(* CoDeSys 2.3.9.25 project: 1.pro *)
(* Libraries: ifm_CR0200\ifm_CR0200_DUMMY_V060002.lib 18.5.06 14:18:58, D:\program files\ifm electronic\CoDeSys V2.3\Targets\ifm\Library\ifm_hydraulic_16bitOS04_V010001.lib 23.10.09 15:40:02, ifm_CR0200\ifm_CR0200_V060003.lib 5.11.09 16:13:42, standard.lib 4.10.05 11:14:46, SysLibCallback.lib 5.6.03 00:36:48, 3S_CANopenManagerOptTableEx.lib 16.7.10 11:11:06, 3S_CanDrvOptTableEx.lib 16.7.10 11:11:16, 3S_CANopenNetVarOptTableEx.lib 16.7.10 11:11:26, Util.lib 6.11.07 14:39:24, ifm_CR0200\ifm_CR0200_CANopenMaster_V040003.lib 7.2.07 16:08:18, 3S_CANopenMasterOptTableEx.lib 16.7.10 11:11:12 *)

(* PLC configuration (modules and I/O channels)
Inputs/Outputs [CR0200] node 0, in %IB0 out %QB0
  Inputs Port0 [Eingangsport0] node 0, in %IB0 out %QB0
    I00 AT %IX0.0 [BoolChannelIn] Connector 1, Pin 08, (see Configuration Byte I00_MODE)
    I01 AT %IX0.1 [BoolChannelIn] Connector 1, Pin 27, (see Configuration Byte I01_MODE)
    I02 AT %IX0.2 [BoolChannelIn] Connector 1, Pin 09, (see Configuration Byte I02_MODE)
    I03 AT %IX0.3 [BoolChannelIn] Connector 1, Pin 28, (see Configuration Byte I03_MODE)
    I04 AT %IX0.4 [BoolChannelIn] Connector 1, Pin 10, (see Configuration Byte I04_MODE)
    I05 AT %IX0.5 [BoolChannelIn] Connector 1, Pin 29, (see Configuration Byte I05_MODE)
    I06 AT %IX0.6 [BoolChannelIn] Connector 1, Pin 11, (see Configuration Byte I06_MODE)
    I07 AT %IX0.7 [BoolChannelIn] Connector 1, Pin 30, (see Configuration Byte I07_MODE)
  Inputs Port1 [Eingangsport1] node 0, in %IB1 out %QB0
    I10 AT %IX0.8 [BoolChannelIn] Connector 1, Pin 44, (see Configuration Byte I10_MODE)
    I11 AT %IX0.9 [BoolChannelIn] Connector 1, Pin 45, (see Configuration Byte I11_MODE)
    I12 AT %IX0.10 [BoolChannelIn] Connector 1, Pin 46, (see Configuration Byte I12_MODE)
    I13 AT %IX0.11 [BoolChannelIn] Connector 1, Pin 47, (see Configuration Byte I13_MODE)
    I14 AT %IX0.12 [BoolChannelIn] Connector 1, Pin 20, (see Configuration Byte I14_MODE)
    I15 AT %IX0.13 [BoolChannelIn] Connector 1, Pin 02, (see Configuration Byte I15_MODE)
    I16 AT %IX0.14 [BoolChannelIn] Connector 1, Pin 21, (see Configuration Byte I16_MODE)
    I17 AT %IX0.15 [BoolChannelIn] Connector 1, Pin 38, (see Configuration Byte I17_MODE)
  Inputs Port2 [Eingangsport2] node 0, in %IB2 out %QB0
    I20 AT %IX1.0 [BoolChannelIn] Connector 1, Pin 36, (see Configuration Byte I20_MODE)
    I21 AT %IX1.1 [BoolChannelIn] Connector 1, Pin 54, (see Configuration Byte I21_MODE)
    I22 AT %IX1.2 [BoolChannelIn] Connector 1, Pin 17, (see Configuration Byte I22_MODE)
    I23 AT %IX1.3 [BoolChannelIn] Connector 1, Pin 53, (see Configuration Byte I23_MODE)
    I24 AT %IX1.4 [BoolChannelIn] Connector 1, Pin 19, (see Configuration Byte I24_MODE)
    I25 AT %IX1.5 [BoolChannelIn] Connector 1, Pin 55, (see Configuration Byte I25_MODE)
    I26 AT %IX1.6 [BoolChannelIn] Connector 1, Pin 18, (see Configuration Byte I26_MODE)
    I27 AT %IX1.7 [BoolChannelIn] Connector 1, Pin 37, (see Configuration Byte I27_MODE)
  Inputs Port3 [Eingangsport3] node 0, in %IB3 out %QB0
    I30 AT %IX1.8 [BoolChannelIn] Connector 1, Pin 39, (see Configuration Byte I30_MODE)
    I31 AT %IX1.9 [BoolChannelIn] Connector 1, Pin 03, (see Configuration Byte I31_MODE)
    I32 AT %IX1.10 [BoolChannelIn] Connector 1, Pin 40, (see Configuration Byte I32_MODE)
    I33 AT %IX1.11 [BoolChannelIn] Connector 1, Pin 22, (see Configuration Byte I33_MODE)
    I34 AT %IX1.12 [BoolChannelIn] Connector 1, Pin 41, (see Configuration Byte I34_MODE)
    I35 AT %IX1.13 [BoolChannelIn] Connector 1, Pin 42, (see Configuration Byte I35_MODE)
    I36 AT %IX1.14 [BoolChannelIn] Connector 1, Pin 43, (see Configuration Byte I36_MODE)
    I37 AT %IX1.15 [BoolChannelIn] Connector 1, Pin 04, (see Configuration Byte I37_MODE)
  Inputs Port4 [Eingangsport4] node 0, in %IB4 out %QB0
    I40 AT %IX2.0 [BoolChannelIn] Connector 1, Pin 48, (see Configuration Byte I40_MODE)
    I41 AT %IX2.1 [BoolChannelIn] Connector 1, Pin 49, (see Configuration Byte I41_MODE)
    I42 AT %IX2.2 [BoolChannelIn] Connector 1, Pin 31, (see Configuration Byte I42_MODE)
    I43 AT %IX2.3 [BoolChannelIn] Connector 1, Pin 50, (see Configuration Byte I43_MODE)
    I44 AT %IX2.4 [BoolChannelIn] Connector 1, Pin 51, (see Configuration Byte I44_MODE)
    I45 AT %IX2.5 [BoolChannelIn] Connector 1, Pin 52, (see Configuration Byte I45_MODE)
    I46 AT %IX2.6 [BoolChannelIn] Connector 1, Pin 16, (see Configuration Byte I46_MODE)
    I47 AT %IX2.7 [BoolChannelIn] Connector 1, Pin 35, (see Configuration Byte I47_MODE)
  Inputs Analog [Analogport] node 0, in %IB6 out %QB0
    ANALOG0 AT %IW3 [WordChannelIn] Connector 1, Pin 08, ANALOG CHANNEL 0
    ANALOG1 AT %IW4 [WordChannelIn] Connector 1, Pin 27, ANALOG CHANNEL 1
    ANALOG2 AT %IW5 [WordChannelIn] Connector 1, Pin 09, ANALOG CHANNEL 2
    ANALOG3 AT %IW6 [WordChannelIn] Connector 1, Pin 28, ANALOG CHANNEL 3
    ANALOG4 AT %IW7 [WordChannelIn] Connector 1, Pin 10, ANALOG CHANNEL 4
    ANALOG5 AT %IW8 [WordChannelIn] Connector 1, Pin 29, ANALOG CHANNEL 5
    ANALOG6 AT %IW9 [WordChannelIn] Connector 1, Pin 11, ANALOG CHANNEL 6
    ANALOG7 AT %IW10 [WordChannelIn] Connector 1, Pin 30, ANALOG CHANNEL 7
  Inputs Miscellaneous [Eingaenge] node 0, in %IB22 out %QB0
    SUPPLY_VOLTAGE AT %IW11 [WordChannelIn] SUPPLY VOLTAGE
    CLAMP_15 AT %IX12.0 [WordChannelIn] CLAMP 15
  Outputs Port1 [Ausgangsport1] node 0, in %IB64 out %QB0
    Q10 AT %QX0.0 [BoolChannelOut] Connector 1, Pin 44, (see Configuration Byte Q10_MODE)
    Q11 AT %QX0.1 [BoolChannelOut] Connector 1, Pin 45, (see Configuration Byte Q11_MODE)
    Q12 AT %QX0.2 [BoolChannelOut] Connector 1, Pin 46, (see Configuration Byte Q12_MODE)
    Q13 AT %QX0.3 [BoolChannelOut] Connector 1, Pin 47, (see Configuration Byte Q13_MODE)
  Outputs Port2 [Ausgangsport2] node 0, in %IB64 out %QB0
    Q20 AT %QX0.4 [BoolChannelOut] Connector 1, Pin 36, (see Configuration Byte Q20_MODE)
    Q21 AT %QX0.5 [BoolChannelOut] Connector 1, Pin 54, (see Configuration Byte Q21_MODE)
    Q22 AT %QX0.6 [BoolChannelOut] Connector 1, Pin 17, (see Configuration Byte Q22_MODE)
    Q23 AT %QX0.7 [BoolChannelOut] Connector 1, Pin 53, (see Configuration Byte Q23_MODE)
  Outputs Port3 [Ausgangsport3] node 0, in %IB64 out %QB1
    Q30 AT %QX0.8 [BoolChannelOut] Connector 1, Pin 39, (see Configuration Byte Q30_MODE)
    Q31 AT %QX0.9 [BoolChannelOut] Connector 1, Pin 03, (see Configuration Byte Q31_MODE)
    Q32 AT %QX0.10 [BoolChannelOut] Connector 1, Pin 40, (see Configuration Byte Q32_MODE)
    Q33 AT %QX0.11 [BoolChannelOut] Connector 1, Pin 22, (see Configuration Byte Q33_MODE)
    Q34 AT %QX0.12 [BoolChannelOut] Connector 1, Pin 41, (see Configuration Byte Q34_MODE)
    Q35 AT %QX0.13 [BoolChannelOut] Connector 1, Pin 42, (see Configuration Byte Q35_MODE)
    Q36 AT %QX0.14 [BoolChannelOut] Connector 1, Pin 43, (see Configuration Byte Q36_MODE)
    Q37 AT %QX0.15 [BoolChannelOut] Connector 1, Pin 04, (see Configuration Byte Q37_MODE)
  Outputs Port4 [Ausgangsport4] node 0, in %IB64 out %QB2
    Q40 AT %QX1.0 [BoolChannelOut] Connector 1, Pin 48, (see Configuration Byte Q40_MODE)
    Q41 AT %QX1.1 [BoolChannelOut] Connector 1, Pin 49, (see Configuration Byte Q41_MODE)
    Q42 AT %QX1.2 [BoolChannelOut] Connector 1, Pin 31, (see Configuration Byte Q42_MODE)
    Q43 AT %QX1.3 [BoolChannelOut] Connector 1, Pin 50, (see Configuration Byte Q43_MODE)
    Q44 AT %QX1.4 [BoolChannelOut] Connector 1, Pin 51, (see Configuration Byte Q44_MODE)
    Q45 AT %QX1.5 [BoolChannelOut] Connector 1, Pin 52, (see Configuration Byte Q45_MODE)
    Q46 AT %QX1.6 [BoolChannelOut] Connector 1, Pin 16, (see Configuration Byte Q46_MODE)
    Q47 AT %QX1.7 [BoolChannelOut] Connector 1, Pin 35, (see Configuration Byte Q47_MODE)
  Input Modes Port0 [EingangsModi0] node 0, in %IB64 out %QB8
    I00_MODE AT %QB8 [ByteChannelOut] Configuration Byte for Input Pin 08, Connector 1
    I01_MODE AT %QB9 [ByteChannelOut] Configuration Byte for Input Pin 27, Connector 1
    I02_MODE AT %QB10 [ByteChannelOut] Configuration Byte for Input Pin 09, Connector 1
    I03_MODE AT %QB11 [ByteChannelOut] Configuration Byte for Input Pin 28, Connector 1
    I04_MODE AT %QB12 [ByteChannelOut] Configuration Byte for Input Pin 10, Connector 1
    I05_MODE AT %QB13 [ByteChannelOut] Configuration Byte for Input Pin 29, Connector 1
    I06_MODE AT %QB14 [ByteChannelOut] Configuration Byte for Input Pin 11, Connector 1
    I07_MODE AT %QB15 [ByteChannelOut] Configuration Byte for Input Pin 30, Connector 1
  Input Modes Port1 [EingangsModi1] node 0, in %IB64 out %QB16
    I14_MODE AT %QB16 [ByteChannelOut] Configuration Byte for Input Pin 20, Connector 1
    I15_MODE AT %QB17 [ByteChannelOut] Configuration Byte for Input Pin 02, Connector 1
    I16_MODE AT %QB18 [ByteChannelOut] Configuration Byte for Input Pin 21, Connector 1
    I17_MODE AT %QB19 [ByteChannelOut] Configuration Byte for Input Pin 38, Connector 1
  Input Modes Port2 [EingangsModi2] node 0, in %IB64 out %QB20
    I24_MODE AT %QB20 [ByteChannelOut] Configuration Byte for Input Pin 19, Connector 1
    I25_MODE AT %QB21 [ByteChannelOut] Configuration Byte for Input Pin 55, Connector 1
    I26_MODE AT %QB22 [ByteChannelOut] Configuration Byte for Input Pin 18, Connector 1
    I27_MODE AT %QB23 [ByteChannelOut] Configuration Byte for Input Pin 37, Connector 1
  Input Modes Port3 [EingangsModi3] node 0, in %IB64 out %QB24
    I30_MODE AT %QB24 [ByteChannelOut] Configuration Byte for Input Pin 39, Connector 1
    I31_MODE AT %QB25 [ByteChannelOut] Configuration Byte for Input Pin 03, Connector 1
    I32_MODE AT %QB26 [ByteChannelOut] Configuration Byte for Input Pin 40, Connector 1
    I33_MODE AT %QB27 [ByteChannelOut] Configuration Byte for Input Pin 22, Connector 1
    I34_MODE AT %QB28 [ByteChannelOut] Configuration Byte for Input Pin 41, Connector 1
    I35_MODE AT %QB29 [ByteChannelOut] Configuration Byte for Input Pin 42, Connector 1
    I36_MODE AT %QB30 [ByteChannelOut] Configuration Byte for Input Pin 43, Connector 1
    I37_MODE AT %QB31 [ByteChannelOut] Configuration Byte for Input Pin 04, Connector 1
  Input Modes Port4 [EingangsModi4] node 0, in %IB64 out %QB32
    I40_MODE AT %QB32 [ByteChannelOut] Configuration Byte for Input Pin 48, Connector 1
    I41_MODE AT %QB33 [ByteChannelOut] Configuration Byte for Input Pin 49, Connector 1
    I42_MODE AT %QB34 [ByteChannelOut] Configuration Byte for Input Pin 31, Connector 1
    I43_MODE AT %QB35 [ByteChannelOut] Configuration Byte for Input Pin 50, Connector 1
    I44_MODE AT %QB36 [ByteChannelOut] Configuration Byte for Input Pin 51, Connector 1
    I45_MODE AT %QB37 [ByteChannelOut] Configuration Byte for Input Pin 52, Connector 1
    I46_MODE AT %QB38 [ByteChannelOut] Configuration Byte for Input Pin 16, Connector 1
    I47_MODE AT %QB39 [ByteChannelOut] Configuration Byte for Input Pin 35, Connector 1
  Output Modes Port1 [AusgangsModi1] node 0, in %IB64 out %QB40
    Q10_MODE AT %QB40 [ByteChannelOut] Configuration Byte for Output Pin 44, Connector 1
    Q11_MODE AT %QB41 [ByteChannelOut] Configuration Byte for Output Pin 45, Connector 1
    Q12_MODE AT %QB42 [ByteChannelOut] Configuration Byte for Output Pin 46, Connector 1
    Q13_MODE AT %QB43 [ByteChannelOut] Configuration Byte for Output Pin 47, Connector 1
  Output Modes Port2 [AusgangsModi2] node 0, in %IB64 out %QB44
    Q20_MODE AT %QB44 [ByteChannelOut] Configuration Byte for Output Pin 36, Connector 1
    Q21_MODE AT %QB45 [ByteChannelOut] Configuration Byte for Output Pin 54, Connector 1
    Q22_MODE AT %QB46 [ByteChannelOut] Configuration Byte for Output Pin 17, Connector 1
    Q23_MODE AT %QB47 [ByteChannelOut] Configuration Byte for Output Pin 53, Connector 1
  Output Modes Port3 [AusgangsModi3] node 0, in %IB64 out %QB48
    Q30_MODE AT %QB48 [ByteChannelOut] Configuration Byte for Output Pin 39, Connector 1
    Q31_MODE AT %QB49 [ByteChannelOut] Configuration Byte for Output Pin 03, Connector 1
    Q32_MODE AT %QB50 [ByteChannelOut] Configuration Byte for Output Pin 40, Connector 1
    Q33_MODE AT %QB51 [ByteChannelOut] Configuration Byte for Output Pin 22, Connector 1
    Q34_MODE AT %QB52 [ByteChannelOut] Configuration Byte for Output Pin 41, Connector 1
    Q35_MODE AT %QB53 [ByteChannelOut] Configuration Byte for Output Pin 42, Connector 1
    Q36_MODE AT %QB54 [ByteChannelOut] Configuration Byte for Output Pin 43, Connector 1
    Q37_MODE AT %QB55 [ByteChannelOut] Configuration Byte for Output Pin 04, Connector 1
  Output Modes Port4 [AusgangsModi4] node 0, in %IB64 out %QB56
    Q40_MODE AT %QB56 [ByteChannelOut] Configuration Byte for Output Pin 48, Connector 1
    Q41_MODE AT %QB57 [ByteChannelOut] Configuration Byte for Output Pin 49, Connector 1
    Q42_MODE AT %QB58 [ByteChannelOut] Configuration Byte for Output Pin 31, Connector 1
    Q43_MODE AT %QB59 [ByteChannelOut] Configuration Byte for Output Pin 50, Connector 1
    Q44_MODE AT %QB60 [ByteChannelOut] Configuration Byte for Output Pin 51, Connector 1
    Q45_MODE AT %QB61 [ByteChannelOut] Configuration Byte for Output Pin 52, Connector 1
    Q46_MODE AT %QB62 [ByteChannelOut] Configuration Byte for Output Pin 16, Connector 1
    Q47_MODE AT %QB63 [ByteChannelOut] Configuration Byte for Output Pin 35, Connector 1
Extended Inputs Port0 [Eingangsport0E] node 0, in %IB64 out %QB64
  I00_E AT %IX32.0 [BoolChannelIn] Connector 2, Pin 08, (see Configuration Byte I00_MODE_E)
  I01_E AT %IX32.1 [BoolChannelIn] Connector 2, Pin 27, (see Configuration Byte I01_MODE_E)
  I02_E AT %IX32.2 [BoolChannelIn] Connector 2, Pin 09, (see Configuration Byte I02_MODE_E)
  I03_E AT %IX32.3 [BoolChannelIn] Connector 2, Pin 28, (see Configuration Byte I03_MODE_E)
  I04_E AT %IX32.4 [BoolChannelIn] Connector 2, Pin 10, (see Configuration Byte I04_MODE_E)
  I05_E AT %IX32.5 [BoolChannelIn] Connector 2, Pin 29, (see Configuration Byte I05_MODE_E)
  I06_E AT %IX32.6 [BoolChannelIn] Connector 2, Pin 11, (see Configuration Byte I06_MODE_E)
  I07_E AT %IX32.7 [BoolChannelIn] Connector 2, Pin 30, (see Configuration Byte I07_MODE_E)
Extended Inputs Port1 [Eingangsport1E] node 0, in %IB65 out %QB64
  I10_E AT %IX32.8 [BoolChannelIn] Connector 2, Pin 44, (see Configuration Byte I10_MODE_E)
  I11_E AT %IX32.9 [BoolChannelIn] Connector 2, Pin 45, (see Configuration Byte I11_MODE_E)
  I12_E AT %IX32.10 [BoolChannelIn] Connector 2, Pin 46, (see Configuration Byte I12_MODE_E)
  I13_E AT %IX32.11 [BoolChannelIn] Connector 2, Pin 47, (see Configuration Byte I13_MODE_E)
  I14_E AT %IX32.12 [BoolChannelIn] Connector 2, Pin 20, (see Configuration Byte I14_MODE_E)
  I15_E AT %IX32.13 [BoolChannelIn] Connector 2, Pin 02, (see Configuration Byte I15_MODE_E)
  I16_E AT %IX32.14 [BoolChannelIn] Connector 2, Pin 21, (see Configuration Byte I16_MODE_E)
  I17_E AT %IX32.15 [BoolChannelIn] Connector 2, Pin 38, (see Configuration Byte I17_MODE_E)
I20_E AT %IX33.0 [BoolChannelIn] Connector 2, Pin 36, (see Configuration Byte I20_MODE_E)
I21_E AT %IX33.1 [BoolChannelIn] Connector 2, Pin 54, (see Configuration Byte I21_MODE_E)
I22_E AT %IX33.2 [BoolChannelIn] Connector 2, Pin 17, (see Configuration Byte I22_MODE_E)
I23_E AT %IX33.3 [BoolChannelIn] Connector 2, Pin 53, (see Configuration Byte I23_MODE_E)
I24_E AT %IX33.4 [BoolChannelIn] Connector 2, Pin 19, (see Configuration Byte I24_MODE_E)
I25_E AT %IX33.5 [BoolChannelIn] Connector 2, Pin 55, (see Configuration Byte I25_MODE_E)
I26_E AT %IX33.6 [BoolChannelIn] Connector 2, Pin 18, (see Configuration Byte I26_MODE_E)
I27_E AT %IX33.7 [BoolChannelIn] Connector 2, Pin 37, (see Configuration Byte I27_MODE_E)
I30_E AT %IX33.8 [BoolChannelIn] Connector 2, Pin 39, (see Configuration Byte I30_MODE_E)
I31_E AT %IX33.9 [BoolChannelIn] Connector 2, Pin 03, (see Configuration Byte I31_MODE_E)
I32_E AT %IX33.10 [BoolChannelIn] Connector 2, Pin 40, (see Configuration Byte I32_MODE_E)
I33_E AT %IX33.11 [BoolChannelIn] Connector 2, Pin 22, (see Configuration Byte I33_MODE_E)
I34_E AT %IX33.12 [BoolChannelIn] Connector 2, Pin 41, (see Configuration Byte I34_MODE_E)
I35_E AT %IX33.13 [BoolChannelIn] Connector 2, Pin 42, (see Configuration Byte I35_MODE_E)
I36_E AT %IX33.14 [BoolChannelIn] Connector 2, Pin 43, (see Configuration Byte I36_MODE_E)
I37_E AT %IX33.15 [BoolChannelIn] Connector 2, Pin 04, (see Configuration Byte I37_MODE_E)
Extended Inputs Port4 [Eingangsport4E] node 0, in %IB68 out %QB64
  I40_E AT %IX34.0 [BoolChannelIn] Connector 2, Pin 48, (see Configuration Byte I40_MODE_E)
  I41_E AT %IX34.1 [BoolChannelIn] Connector 2, Pin 49, (see Configuration Byte I41_MODE_E)
  I42_E AT %IX34.2 [BoolChannelIn] Connector 2, Pin 31, (see Configuration Byte I42_MODE_E)
  I43_E AT %IX34.3 [BoolChannelIn] Connector 2, Pin 50, (see Configuration Byte I43_MODE_E)
  I44_E AT %IX34.4 [BoolChannelIn] Connector 2, Pin 51, (see Configuration Byte I44_MODE_E)
  I45_E AT %IX34.5 [BoolChannelIn] Connector 2, Pin 52, (see Configuration Byte I45_MODE_E)
  I46_E AT %IX34.6 [BoolChannelIn] Connector 2, Pin 16, (see Configuration Byte I46_MODE_E)
  I47_E AT %IX34.7 [BoolChannelIn] Connector 2, Pin 35, (see Configuration Byte I47_MODE_E)
Extended Inputs Analog [AnalogportE] node 0, in %IB70 out %QB64
  ANALOG0_E AT %IW35 [WordChannelIn] Connector 2, Pin 08, ANALOG CHANNEL 0
  ANALOG1_E AT %IW36 [WordChannelIn] Connector 2, Pin 27, ANALOG CHANNEL 1
  ANALOG2_E AT %IW37 [WordChannelIn] Connector 2, Pin 09, ANALOG CHANNEL 2
  ANALOG3_E AT %IW38 [WordChannelIn] Connector 2, Pin 28, ANALOG CHANNEL 3
  ANALOG4_E AT %IW39 [WordChannelIn] Connector 2, Pin 10, ANALOG CHANNEL 4
  ANALOG5_E AT %IW40 [WordChannelIn] Connector 2, Pin 29, ANALOG CHANNEL 5
  ANALOG6_E AT %IW41 [WordChannelIn] Connector 2, Pin 11, ANALOG CHANNEL 6
  ANALOG7_E AT %IW42 [WordChannelIn] Connector 2, Pin 30, ANALOG CHANNEL 7
Extended Inputs Miscellaneous [EingaengeE] node 0, in %IB86 out %QB64
  SUPPLY_VOLTAGE_E AT %IW43 [WordChannelIn] SUPPLY VOLTAGE
  CLAMP_15_E AT %IX44.0 [WordChannelIn] CLAMP 15
Extended Outputs Port1 [Ausgangsport1E] node 0, in %IB128 out %QB64
  Q10_E AT %QX32.0 [BoolChannelOut] Connector 2, Pin 44, (see Configuration Byte Q10_MODE_E)
  Q11_E AT %QX32.1 [BoolChannelOut] Connector 2, Pin 45, (see Configuration Byte Q11_MODE_E)
  Q12_E AT %QX32.2 [BoolChannelOut] Connector 2, Pin 46, (see Configuration Byte Q11_MODE_E)
  Q13_E AT %QX32.3 [BoolChannelOut] Connector 2, Pin 47, (see Configuration Byte Q11_MODE_E)
Extended Outputs Port2 [Ausgangsport2E] node 0, in %IB128 out %QB64
  Q20_E AT %QX32.4 [BoolChannelOut] Connector 2, Pin 36, (see Configuration Byte Q20_MODE_E)
  Q21_E AT %QX32.5 [BoolChannelOut] Connector 2, Pin 54, (see Configuration Byte Q21_MODE_E)
  Q22_E AT %QX32.6 [BoolChannelOut] Connector 2, Pin 17, (see Configuration Byte Q22_MODE_E)
  Q23_E AT %QX32.7 [BoolChannelOut] Connector 2, Pin 53, (see Configuration Byte Q23_MODE_E)
Q30_E AT %QX32.8 [BoolChannelOut] Connector 2, Pin 39, (see Configuration Byte Q30_MODE_E)
Q31_E AT %QX32.9 [BoolChannelOut] Connector 2, Pin 03, (see Configuration Byte Q31_MODE_E)
Q32_E AT %QX32.10 [BoolChannelOut] Connector 2, Pin 40, (see Configuration Byte Q32_MODE_E)
Q33_E AT %QX32.11 [BoolChannelOut] Connector 2, Pin 22, (see Configuration Byte Q33_MODE_E)
Q34_E AT %QX32.12 [BoolChannelOut] Connector 2, Pin 41, (see Configuration Byte Q34_MODE_E)
Q35_E AT %QX32.13 [BoolChannelOut] Connector 2, Pin 42, (see Configuration Byte Q35_MODE_E)
Q36_E AT %QX32.14 [BoolChannelOut] Connector 2, Pin 43, (see Configuration Byte Q36_MODE_E)
Q37_E AT %QX32.15 [BoolChannelOut] Connector 2, Pin 04, (see Configuration Byte Q37_MODE_E)
Extended Outputs Port4 [Ausgangsport4E] node 0, in %IB128 out %QB66
  Q40_E AT %QX33.0 [BoolChannelOut] Connector 2, Pin 48, (see Configuration Byte Q40_MODE_E)
  Q41_E AT %QX33.1 [BoolChannelOut] Connector 2, Pin 49, (see Configuration Byte Q41_MODE_E)
  Q42_E AT %QX33.2 [BoolChannelOut] Connector 2, Pin 31, (see Configuration Byte Q42_MODE_E)
  Q43_E AT %QX33.3 [BoolChannelOut] Connector 2, Pin 50, (see Configuration Byte Q43_MODE_E)
  Q44_E AT %QX33.4 [BoolChannelOut] Connector 2, Pin 51, (see Configuration Byte Q44_MODE_E)
  Q45_E AT %QX33.5 [BoolChannelOut] Connector 2, Pin 52, (see Configuration Byte Q45_MODE_E)
  Q46_E AT %QX33.6 [BoolChannelOut] Connector 2, Pin 16, (see Configuration Byte Q46_MODE_E)
  Q47_E AT %QX33.7 [BoolChannelOut] Connector 2, Pin 35, (see Configuration Byte Q47_MODE_E)
Extended Input Modes Port0 [EingangsModi0E] node 0, in %IB128 out %QB72
  I00Mode_E AT %QB72 [ByteChannelOut] Configuration Byte for Input Pin 08, Connector 2
  I01Mode_E AT %QB73 [ByteChannelOut] Configuration Byte for Input Pin 27, Connector 2
  I02Mode_E AT %QB74 [ByteChannelOut] Configuration Byte for Input Pin 09, Connector 2
  I03Mode_E AT %QB75 [ByteChannelOut] Configuration Byte for Input Pin 28, Connector 2
  I04Mode_E AT %QB76 [ByteChannelOut] Configuration Byte for Input Pin 10, Connector 2
  I05Mode_E AT %QB77 [ByteChannelOut] Configuration Byte for Input Pin 29, Connector 2
  I06Mode_E AT %QB78 [ByteChannelOut] Configuration Byte for Input Pin 11, Connector 2
  I07Mode_E AT %QB79 [ByteChannelOut] Configuration Byte for Input Pin 30, Connector 2
Extended Input Modes Port1 [EingangsModi1E] node 0, in %IB128 out %QB80
  I14Mode_E AT %QB80 [ByteChannelOut] Configuration Byte for Input Pin 20, Connector 2
  I15Mode_E AT %QB81 [ByteChannelOut] Configuration Byte for Input Pin 02, Connector 2
  I16Mode_E AT %QB82 [ByteChannelOut] Configuration Byte for Input Pin 21, Connector 2
  I17Mode_E AT %QB83 [ByteChannelOut] Configuration Byte for Input Pin 38, Connector 2
Extended Input Modes Port2 [EingangsModi2E] node 0, in %IB128 out %QB84
  I24Mode_E AT %QB84 [ByteChannelOut] Configuration Byte for Input Pin 19, Connector 2
  I25Mode_E AT %QB85 [ByteChannelOut] Configuration Byte for Input Pin 55, Connector 2
  I26Mode_E AT %QB86 [ByteChannelOut] Configuration Byte for Input Pin 18, Connector 2
  I27Mode_E AT %QB87 [ByteChannelOut] Configuration Byte for Input Pin 37, Connector 2
Extended Input Modes Port3 [EingangsModi3E] node 0, in %IB128 out %QB88
  I30Mode_E AT %QB88 [ByteChannelOut] Configuration Byte for Input Pin 39, Connector 2
  I31Mode_E AT %QB89 [ByteChannelOut] Configuration Byte for Input Pin 03, Connector 2
  I32Mode_E AT %QB90 [ByteChannelOut] Configuration Byte for Input Pin 40, Connector 2
  I33Mode_E AT %QB91 [ByteChannelOut] Configuration Byte for Input Pin 22, Connector 2
  I34Mode_E AT %QB92 [ByteChannelOut] Configuration Byte for Input Pin 41, Connector 2
  I35Mode_E AT %QB93 [ByteChannelOut] Configuration Byte for Input Pin 42, Connector 2
  I36Mode_E AT %QB94 [ByteChannelOut] Configuration Byte for Input Pin 43, Connector 2
  I37Mode_E AT %QB95 [ByteChannelOut] Configuration Byte for Input Pin 04, Connector 2
Extended Input Modes Port4 [EingangsModi4E] node 0, in %IB128 out %QB96
  I40Mode_E AT %QB96 [ByteChannelOut] Configuration Byte for Input Pin 48, Connector 2
  I41Mode_E AT %QB97 [ByteChannelOut] Configuration Byte for Input Pin 49, Connector 2
  I42Mode_E AT %QB98 [ByteChannelOut] Configuration Byte for Input Pin 31, Connector 2
  I43Mode_E AT %QB99 [ByteChannelOut] Configuration Byte for Input Pin 50, Connector 2
  I44Mode_E AT %QB100 [ByteChannelOut] Configuration Byte for Input Pin 51, Connector 2
  I45Mode_E AT %QB101 [ByteChannelOut] Configuration Byte for Input Pin 52, Connector 2
  I46Mode_E AT %QB102 [ByteChannelOut] Configuration Byte for Input Pin 16, Connector 2
  I47Mode_E AT %QB103 [ByteChannelOut] Configuration Byte for Input Pin 35, Connector 2
Extended Output Modes Port1 [AusgangsModi1E] node 0, in %IB128 out %QB104
  Q10Mode_E AT %QB104 [ByteChannelOut] Configuration Byte for Output Pin 44, Connector 2
  Q11Mode_E AT %QB105 [ByteChannelOut] Configuration Byte for Output Pin 45, Connector 2
  Q12Mode_E AT %QB106 [ByteChannelOut] Configuration Byte for Output Pin 46, Connector 2
  Q13Mode_E AT %QB107 [ByteChannelOut] Configuration Byte for Output Pin 47, Connector 2
Extended Output Modes Port2 [AusgangsModi2E] node 0, in %IB128 out %QB108
  Q20Mode_E AT %QB108 [ByteChannelOut] Configuration Byte for Output Pin 36, Connector 2
  Q21Mode_E AT %QB109 [ByteChannelOut] Configuration Byte for Output Pin 54, Connector 2
  Q22Mode_E AT %QB110 [ByteChannelOut] Configuration Byte for Output Pin 17, Connector 2
  Q23Mode_E AT %QB111 [ByteChannelOut] Configuration Byte for Output Pin 53, Connector 2
Extended Output Modes Port3 [AusgangsModi3E] node 0, in %IB128 out %QB112
  Q30Mode_E AT %QB112 [ByteChannelOut] Configuration Byte for Output Pin 39, Connector 2
  Q31Mode_E AT %QB113 [ByteChannelOut] Configuration Byte for Output Pin 03, Connector 2
  Q32Mode_E AT %QB114 [ByteChannelOut] Configuration Byte for Output Pin 40, Connector 2
  Q33Mode_E AT %QB115 [ByteChannelOut] Configuration Byte for Output Pin 22, Connector 2
  Q34Mode_E AT %QB116 [ByteChannelOut] Configuration Byte for Output Pin 41, Connector 2
  Q35Mode_E AT %QB117 [ByteChannelOut] Configuration Byte for Output Pin 42, Connector 2
  Q36Mode_E AT %QB118 [ByteChannelOut] Configuration Byte for Output Pin 43, Connector 2
  Q37Mode_E AT %QB119 [ByteChannelOut] Configuration Byte for Output Pin 04, Connector 2
Extended Output Modes Port4 [AusgangsModi4E] node 0, in %IB128 out %QB120
  Q40Mode_E AT %QB120 [ByteChannelOut] Configuration Byte for Output Pin 48, Connector 2
  Q41Mode_E AT %QB121 [ByteChannelOut] Configuration Byte for Output Pin 49, Connector 2
  Q42Mode_E AT %QB122 [ByteChannelOut] Configuration Byte for Output Pin 31, Connector 2
  Q43Mode_E AT %QB123 [ByteChannelOut] Configuration Byte for Output Pin 50, Connector 2
  Q44Mode_E AT %QB124 [ByteChannelOut] Configuration Byte for Output Pin 51, Connector 2
  Q45Mode_E AT %QB125 [ByteChannelOut] Configuration Byte for Output Pin 52, Connector 2
  Q46Mode_E AT %QB126 [ByteChannelOut] Configuration Byte for Output Pin 16, Connector 2
  Q47Mode_E AT %QB127 [ByteChannelOut] Configuration Byte for Output Pin 35, Connector 2
CR0200, CANopen Master [CanMaster] node 2, in %IB192 out %QB192
*)

(* Global variable list: alarm/alarm_text *)
VAR_GLOBAL

	mv_alarm10001:			BOOL;
	mv_alarm10002:			BOOL;
	mv_alarm10003:			BOOL;
	mv_alarm10004:			BOOL;
	mv_alarm10005: 			BOOL;
	mv_alarm10006: 			BOOL;
	mv_alarm10007: 			BOOL;
	mv_alarm10008:			BOOL;

	mv_alarm10009:			BOOL;
	mv_alarm10010:			BOOL;
	mv_alarm10011:			BOOL;
	mv_alarm10012:			BOOL;
	mv_alarm10013:			BOOL;
	mv_alarm10014: 			BOOL;
	mv_alarm10015: 			BOOL;
	mv_alarm10016: 			BOOL;

	mv_alarm10017:			BOOL;
	mv_alarm10018:			BOOL;
	mv_alarm10019:			BOOL;
	mv_alarm10020:			BOOL;
	mv_alarm10021:			BOOL;
	mv_alarm10022: 			BOOL;
	mv_alarm10023: 			BOOL;
	mv_alarm10024: 			BOOL;

	mv_alarm10025:			BOOL;
	mv_alarm10026:			BOOL;
	mv_alarm10027:			BOOL;
	mv_alarm10028:			BOOL;
	mv_alarm10029:			BOOL;
	mv_alarm10030: 			BOOL;
	mv_alarm10031: 			BOOL;
	mv_alarm10032: 			BOOL;
END_VAR

(* Global variable list: CanOpen implicit Variables *)
VAR_GLOBAL CONSTANT
	MAX_CTRLINDEX : INT := 0;
END_VAR
VAR_GLOBAL CONSTANT
	USE_CANOPEN_NODES : BOOL := FALSE;
	MAX_MASTERINDEX : INT := 0;
	MAX_NODEINDEX : INT := 0;
	MAX_SDOINDEX : INT := 0;
	MAX_PDOINDEX_RX : INT := 0;
	MAX_PDOINDEX_TX : INT := 0;
	MAX_MASTER_ODENTRY_IDX : INT := 0;
END_VAR
VAR_GLOBAL
	pCANopenMaster : ARRAY[0..MAX_MASTERINDEX] OF CanOpenMaster;
	pCanOpenNode : ARRAY[0..MAX_NODEINDEX] OF CanOpenNode;
	pCanOpenSDO : ARRAY[0..MAX_SDOINDEX] OF CanOpenSDO;
	pCanOpenPDO_Rx : ARRAY[0..MAX_PDOINDEX_RX] OF CanOpenPDO_Rx;
	pCanOpenPDO_Tx : ARRAY[0..MAX_PDOINDEX_TX] OF CanOpenPDO_Tx;
	 ODMEntries: ARRAY[0..MAX_MASTER_ODENTRY_IDX] OF CanOpenODEntry;
END_VAR

(* Global variable list: Globale_Variablen *)
VAR_GLOBAL RETAIN
	leveled							:BOOL:=0;
(***通用版程序选择***)
(*
	YT32		10000
	YT32A		10001
	YT32B		10002
	YT32C		10003
	YT32D		10004
	YT32E		10005
	YT32F		10006
	YT32G		10007
	YT32H		10008
	YT32I		10009
	YT32J		10010
	YT32K		10011
	YT32L		10012
	YT32M		10013
	YT32N		10014
	YT32O		10015
	YT32P		10016
	YT32Q		10017
	YT32R		10018
	YT32S		10019
	YT32T		10020
*)
	vehicle_styel					: INT:=10012;
END_VAR

VAR_GLOBAL
	Code_1key					:BOOL;
	Speed_value					:BYTE;
	speed_l						:BOOL;
	encod_sign					: BYTE;
	encod_udint					: UDINT;
	turn_desk_angle				: INT;
(***全局变量***)
	boot_set						: BOOL;
	frequ_set						:BOOL:=1;
	valve_act						: BOOL;

	head_f							:BOOL;
	head_b						:BOOL;
	head_f2						:BOOL;
	head_b2						:BOOL;
	head_f3						:BOOL;
	head_b3						:BOOL;

	auto_extend_triger				: BOOL;
	auto_drawback_triger				: BOOL;

	work_speed_l					:INT;
	work_speed_h				:INT;
	low_speed_l					:INT;
	low_speed_h					:INT;
	high_speed_l					:INT;
	high_speed_h				:INT;

	cruise_sign_set				:BOOL;

	angle_danger01				: INT :=500;
	angle_danger02				: INT := 1500;

	init_1							: BOOL:=TRUE;
	extend_step					:INT;
	withdraw_step				: INT;

	angle_x_offset 				AT%MW0		:INT:=952;
	angle_y_offset 				AT%MW2		:INT:=1039;
	water_height_sign_L 			AT%MW4		: INT:=480;
	water_height_sign_H 		AT%MW6		: INT:=1557;
	oil_pressure_0				AT%MW8		: INT:=4000;
	oil_pressure_22				AT%MW10		: INT:=13931;
	foam_height_sign_L			AT%MW12		: INT:=480;
	foam_height_sign_H			AT%MW14		: INT:=1557;
	water_pressure_0			AT%MW16		: INT:=4000;
	water_pressure_6			AT%MW18		: INT:=6300;

	extend_do						:BOOL;
	withdraw_do					:BOOL;
	high_speed_set				:BOOL;
	high_speed_set1				:BOOL;


 	 extend_left_lv_triger_act		:BOOL;
	extend_right_lv_triger_act	:BOOL;

	rl_ys							:INT:=8;

	triger_left_ground_for			:INT;

	angle_x_m					: WORD;(*倾角X轴实测*)
	angle_y_m					: WORD;(*倾角Y轴实测*)
	oil_pressure_m				: WORD;(*油压实测*)

(***支腿遥控器变量***)
	remote_manual_alarm				:BOOL;
	remote_not_arm_to_station_alarm	:BOOL;

(***网络变量***)
	speed_m						:REAL;
	down_com_sign				:BOOL;
	beep_signal					:BOOL;

	stage_extend_do				:BOOL;
	stage_draw_do				:BOOL;
(***转台变量***)
	tt_turn_com					:BOOL;
	tt_emergency_pump			:BOOL;

	up_down_switch				:BOOL;
	tt_foot_switch					:BOOL;
	tt_engine_startup				:BOOL;
	tt_engine_stop				:BOOL;
	tt_water_pump_open		 	:BOOL;

	tt_engine_acc					:BOOL;(*发动机加速*)
	tt_engine_dec					:BOOL;(*发动机减速*)

	tt_water_canon_open	 		:BOOL;
	tt_water_canon_close	 	:BOOL;

(***工作斗变量***)
	sudden_pump_button		:BOOL;
	stage_extend_over			:BOOL;
	stage_draw_over				:BOOL;

	stage_foot_switch			:BOOL;
	stage_engine_startup		:BOOL;
	stage_engine_stop			:BOOL;
	stage_water_pump_open	:BOOL;
	stage_com					:BOOL;
	stage_engine_acc			:BOOL;(*发动机加速*)
	stage_engine_dec			:BOOL;(*发动机减速*)
	error1							:BOOL;
	error2							:BOOL;

(***屏幕变量***)

	foam_low_sign_set			:BOOL;
	foam_high_sign_set			:BOOL;
	down_zero_set				:BOOL;
	water_low_sign_set			:BOOL;
	water_high_sign_set			:BOOL;
	oil_low_sign_set				:BOOL;
	oil_high_sign_set				:BOOL;
	water_alarm_c				:BOOL;

END_VAR

(* Global variable list: VEHICLE TYPE/io_Variables *)
VAR_GLOBAL
(*************************************A_INPUT*******************************************)
	angle_x												: INT;		(*倾角X轴*)
	angle_y												: INT;		(*倾角Y轴*)
	angle_x_1												: INT;
	angle_y_1												: INT;
	oil_pressure											: WORD;	(*油压*)
	water_pressure										: WORD;	(*系统水压*)
	water_height_sign									: WORD;	(*水位信号*)
	foam_height_sign									: WORD;	(*泡沫液位信号*)
	water_flux												: WORD;	(*水流量信号*)
	speed_sign											: WORD;	(*速度脉冲*)

(**************************************A_OUTPUT***************************************)
	left_front_desired										: WORD;	(*左前垂直伸*)
	right_front_desired									: WORD;	(*右前垂直伸*)
	left_back_desired										: WORD;	(*左后垂直伸*)
	right_back_desired									: WORD;	(*右后垂直伸*)

	right_front_drawback_desired						: WORD;	(*右前垂直收*)
	left_back_drawback_desired							: WORD;	(*左后垂直收*)
	right_back_drawback_desired						: WORD;	(*右后垂直收*)
	left_front_drawback_desired							: WORD;	(*左前垂直收*)

(*************************************D_INPUT*******************************************)
(***支腿***)
	front_left_Lv_ex_check1		(*AT %IX0.6*)			: BOOL;	(*左前水平伸到位*)
	front_right_Lv_ex_check1		(*AT %IX0.7*)			: BOOL;	(*右前水平伸到位*)
	back_left_Lv_ex_check1		(*AT %IX0.12*)		: BOOL;	(*左后水平伸到位*)
	back_right_Lv_ex_check1	(*AT %IX0.13*)		: BOOL;	(*右后水平伸到位*)
	front_left_urt_ex_check1		(*AT %IX0.14*)		: BOOL;	(*左前垂直伸到位*)
	front_right_urt_ex_check1	(*AT %IX0.15*)		: BOOL;	(*右前垂直伸到位*)
	back_left_urt_ex_check1		(*AT %IX1.4*)			: BOOL;	(*左后垂直伸到位*)
	back_right_urt_ex_check1	(*AT %IX1.5*)			: BOOL;	(*右后垂直伸到位*)

	front_left_Lv_ex_check								: BOOL;	(*左前水平伸到位*)
	front_right_Lv_ex_check								: BOOL;	(*右前水平伸到位*)
	back_left_Lv_ex_check								: BOOL;	(*左后水平伸到位*)
	back_right_Lv_ex_check								: BOOL;	(*右后水平伸到位*)
	front_left_urt_ex_check								: BOOL;	(*左前垂直伸到位*)
	front_right_urt_ex_check								: BOOL;	(*右前垂直伸到位*)
	back_left_urt_ex_check								: BOOL;	(*左后垂直伸到位*)
	back_right_urt_ex_check								: BOOL;	(*右后垂直伸到位*)

	front_left_Lv_drb_check		(*AT %IX32.1*)		: BOOL;	(*左前水平收到位*)
	front_right_Lv_drb_check		(*AT %IX32.2*)		: BOOL;	(*右前水平收到位*)
	back_left_Lv_drb_check		(*AT %IX32.3*)		: BOOL;	(*左后水平收到位*)
	back_right_Lv_drb_check	(*AT %IX32.4*)		: BOOL;	(*右后水平收到位*)
	front_left_urt_drb_check1		(*AT %IX32.5*)		: BOOL;	(*左前垂直收到位*)
	front_right_urt_drb_check1	(*AT %IX32.6*)		: BOOL;	(*右前垂直收到位*)
	back_left_urt_drb_check1	(*AT %IX32.7*)		: BOOL;	(*左后垂直收到位*)
	back_right_urt_drb_check1	(*AT %IX32.12	*)		: BOOL;	(*右后垂直收到位*)

	front_left_urt_drb_check								: BOOL;	(*左前垂直收到位*)
	front_right_urt_drb_check							: BOOL;	(*右前垂直收到位*)
	back_left_urt_drb_check								: BOOL;	(*左后垂直收到位*)
	back_right_urt_drb_check							: BOOL;	(*右后垂直收到位*)

(***底盘***)
	engine_run					(*AT %IX2.2*)			: BOOL;	(*发动机启动*)
	engine_stop					(*AT %IX2.3*)			: BOOL;	(*发动机停止*)
	accelerate_sb					(*AT %IX2.0*)			: BOOL;	(*加速*)
	decelerate_sb					(*AT %IX2.1*)			: BOOL;	(*减速*)

(***操作***)
	tt_forcexx						(*AT %IX34.6*)		: BOOL;	(*转台强制*)
	down_force					(*AT %IX34.7*)		: BOOL;	(*下车强制*)
	auto_manu_choice			(*AT %IX34.1*)		: BOOL;	(*自动/手动*)
	water_pump_run_sb			(*AT %IX1.7*)			: BOOL;	(*消防泵开*)
	standby_pump_check								: BOOL;	(*应急泵*)



	left_side_choice 										: BOOL;	(*左单边*)
	right_side_choice										: BOOL;	(*右单边*)

	level_extend_triger_left								: BOOL;	(*自动伸支腿*)
	level_extend_triger_right								: BOOL;	(*自动伸支腿*)
	auto_extend_triger_left								: BOOL;	(*自动伸支腿*)
	auto_extend_triger_right								: BOOL;	(*自动伸支腿*)
	auto_drawback_triger_left							: BOOL;	(*自动收支腿*)
	auto_drawback_triger_right							: BOOL;	(*自动收支腿*)

	level_extend_triger_left1		(*AT %IX34.2*)		: BOOL;	(*自动伸支腿*)
	level_extend_triger_right1	(*AT %IX34.3*)		: BOOL;	(*自动伸支腿*)
	auto_extend_triger_left1		(*AT %IX33.5*)		: BOOL;	(*自动伸支腿*)
	auto_extend_triger_right1	(*AT %IX33.6*)		: BOOL;	(*自动伸支腿*)
	auto_drawback_triger_left1	(*AT %IX33.7*)		: BOOL;	(*自动收支腿*)
	auto_drawback_triger_right1	(*AT %IX34.0*)		: BOOL;	(*自动收支腿*)


(***检测***)
	arm_to_station				(*AT %IX2.4*)			: BOOL;	(*臂架到位检测*)
	water_pump_check			(*AT %IX33.4*)		: BOOL;	(*水泵取力*)
	left_groud_check1			(*AT %IX34.4*)		: BOOL;	(*车胎离地1*)
	left_groud_check2			(*AT %IX34.5*)		: BOOL;	(*车胎离地2*)
	oil_pump_check										: BOOL;	(*油泵检测*)

(***支腿遥控盒***)
	remote_switch_leg									: BOOL;	(*支腿选择*)
	remote_control_left									: BOOL;	(*支腿左*)
	remote_control_right									: BOOL;	(*支腿右*)
	remote_control_up									: BOOL;	(*支腿上*)
	remote_control_down								: BOOL;	(*支腿下*)
	remote_out_front_left									: BOOL;	(*指示灯左前*)
	remote_out_front_back								: BOOL;	(*指示灯左后*)
	remote_out_right_left									: BOOL;	(*指示灯右前*)
	remote_out_right_back								: BOOL;	(*指示灯右后*)

(*************************************D_OUTPUT*****************************************)
(***支腿***)
	left_front_lv_ex_valve			(*AT %QX32.2*)	 	:  BOOL;	(*左前水平伸*)
	left_back_lv_ex_valve			(*AT %QX32.0*) 		:  BOOL;	(*左后水平伸*)
	right_front_lv_ex_valve		(*AT %QX32.6*)		:  BOOL;	(*右前水平伸*)
	right_back_lv_ex_valve		(*AT %QX32.4*)		:  BOOL;	(*右后水平伸*)
	left_front_lv_drb_valve		(*AT %QX32.3*)	 	:  BOOL;	(*左前水平收*)
	left_back_lv_drb_valve		(*AT %QX32.1*) 		:  BOOL;	(*左后水平收*)
	right_front_lv_drb_valve		(*AT %QX32.7*)		:  BOOL;	(*右前水平收*)
	right_back_lv_drb_valve		(*AT %QX32.5*)		:  BOOL;	(*右后水平收*)

(***底盘***)
	enginer_run_ctl				(*AT %QX0.8*)	 		:  BOOL;	(*启动控制*)
	enginer_stop_ctl				(*AT %QX0.9*)	 		:  BOOL;	(*熄火控制*)
	enginer_acc_ctl				(*AT %QX32.9*)	 	:  BOOL;	(*加速控制*)
	enginer_dec_ctl				(*AT %QX32.10*)	 	:  BOOL;	(*减速控制*)

(***操作***)
	water_pump_ctl				(*AT %QX0.10*)	 	:  BOOL;	(*水泵控制*)
	standby_oil_pump							 		:  BOOL;	(*应急泵*)
	up_valve_ctl					(*AT %QX32.14*)	 	:  BOOL;	(*上车阀*)
	down_valve_ctl				(*AT %QX32.15*) 		:  BOOL;	(*下车阀*)

(***指示***)
	over_level_sign				(*AT %QX0.11*)	 	:  BOOL;	(*坡度超限*)
	triger_left_grd_sign			(*AT %QX0.12*)	 	:  BOOL;	(*支腿离地*)
	alarmer_horn					(*AT %QX32.8*)	 	:  BOOL;	(*警报器*)
	triger_flash					(*AT %QX32.13*)	 	:  BOOL;	(*支腿闪光灯*)
	triger_no_drawback_sign					 		:  BOOL;	(*支腿未全缩指示*)
	leveled_sign											:  BOOL;	(*下车调平指示*)
	water_pump_ctl_sign			(*AT %QX0.10*)	 	:  BOOL;	(*水泵控制指示*)

	canon_valve_open 			 (*AT %QX32.11*)		:  BOOL;(*消防炮气阀检测25E*)
	canon_valve_close			(* AT %QX32.12*)		:  BOOL;(*消防炮气阀检测25E*)

	left_f_lv_ex_over				(*AT %QX0.14*)	 	:  BOOL;	(*左前水平伸到位*)
	left_b_lv_ex_over				(*AT %QX0.15*)	 	:  BOOL;	(*左后水平伸到位*)
	right_f_lv_ex_over				(*AT %QX32.11*)	 	:  BOOL;	(*右前水平伸到位*)
	right_b_lv_ex_over			(*AT %QX32.12*)	 	:  BOOL;	(*右后水平伸到位*)
	up_work_sign											:  BOOL;	(*上车工作指示*)
	down_work_sign										:  BOOL;	(*下车工作指示*)
	under_reset_ctl								 		:  BOOL;	(*底盘复位*)

END_VAR

(* Global variable list: VEHICLE TYPE/io_Variables_10011 *)
VAR_GLOBAL
(*************************************A_INPUT*******************************************)
	angle_x												: INT;		(*倾角X轴*)
	angle_y												: INT;		(*倾角Y轴*)
	angle_x_1												: INT;
	angle_y_1												: INT;
	oil_pressure											: WORD;	(*油压*)
	water_pressure										: WORD;	(*系统水压*)
	water_height_sign									: WORD;	(*水位信号*)
	foam_height_sign									: WORD;	(*泡沫液位信号*)
	water_flux												: WORD;	(*水流量信号*)
	speed_sign											: WORD;	(*速度脉冲*)

(**************************************A_OUTPUT***************************************)
	left_front_desired										: WORD;	(*左前垂直伸*)
	right_front_desired									: WORD;	(*右前垂直伸*)
	left_back_desired										: WORD;	(*左后垂直伸*)
	right_back_desired									: WORD;	(*右后垂直伸*)

	right_front_drawback_desired						: WORD;	(*右前垂直收*)
	left_back_drawback_desired							: WORD;	(*左后垂直收*)
	right_back_drawback_desired						: WORD;	(*右后垂直收*)
	left_front_drawback_desired							: WORD;	(*左前垂直收*)

(*************************************D_INPUT*******************************************)
(***支腿***)
	front_left_Lv_ex_check1		AT %IX0.6				: BOOL;	(*左前水平伸到位*)
	front_right_Lv_ex_check1		AT %IX0.7				: BOOL;	(*右前水平伸到位*)
	back_left_Lv_ex_check1		AT %IX0.12			: BOOL;	(*左后水平伸到位*)
	back_right_Lv_ex_check1	AT %IX0.13			: BOOL;	(*右后水平伸到位*)
	front_left_urt_ex_check1		AT %IX0.14			: BOOL;	(*左前垂直伸到位*)
	front_right_urt_ex_check1	AT %IX0.15			: BOOL;	(*右前垂直伸到位*)
	back_left_urt_ex_check1		AT %IX1.4				: BOOL;	(*左后垂直伸到位*)
	back_right_urt_ex_check1	AT %IX1.5				: BOOL;	(*右后垂直伸到位*)

	front_left_Lv_ex_check								: BOOL;	(*左前水平伸到位*)
	front_right_Lv_ex_check								: BOOL;	(*右前水平伸到位*)
	back_left_Lv_ex_check								: BOOL;	(*左后水平伸到位*)
	back_right_Lv_ex_check								: BOOL;	(*右后水平伸到位*)
	front_left_urt_ex_check								: BOOL;	(*左前垂直伸到位*)
	front_right_urt_ex_check								: BOOL;	(*右前垂直伸到位*)
	back_left_urt_ex_check								: BOOL;	(*左后垂直伸到位*)
	back_right_urt_ex_check								: BOOL;	(*右后垂直伸到位*)

	front_left_Lv_drb_check		AT %IX32.1			: BOOL;	(*左前水平收到位*)
	front_right_Lv_drb_check		AT %IX32.2			: BOOL;	(*右前水平收到位*)
	back_left_Lv_drb_check		AT %IX32.3			: BOOL;	(*左后水平收到位*)
	back_right_Lv_drb_check	AT %IX32.4			: BOOL;	(*右后水平收到位*)
	front_left_urt_drb_check1		AT %IX32.5			: BOOL;	(*左前垂直收到位*)
	front_right_urt_drb_check1	AT %IX32.6			: BOOL;	(*右前垂直收到位*)
	back_left_urt_drb_check1	AT %IX32.7			: BOOL;	(*左后垂直收到位*)
	back_right_urt_drb_check1	AT %IX32.12			: BOOL;	(*右后垂直收到位*)

	front_left_urt_drb_check								: BOOL;	(*左前垂直收到位*)
	front_right_urt_drb_check							: BOOL;	(*右前垂直收到位*)
	back_left_urt_drb_check								: BOOL;	(*左后垂直收到位*)
	back_right_urt_drb_check							: BOOL;	(*右后垂直收到位*)

(***底盘***)
	engine_run					AT %IX2.2				: BOOL;	(*发动机启动*)
	engine_stop					AT %IX2.3				: BOOL;	(*发动机停止*)
	accelerate_sb					AT %IX2.0				: BOOL;	(*加速*)
	decelerate_sb					AT %IX2.1				: BOOL;	(*减速*)

(***操作***)
	tt_forcexx						AT %IX34.6			: BOOL;	(*转台强制*)
	down_force					AT %IX34.7			: BOOL;	(*下车强制*)
	auto_manu_choice			AT %IX34.1			: BOOL;	(*自动/手动*)
	water_pump_run_sb			AT %IX1.7				: BOOL;	(*消防泵开*)
	standby_pump_check								: BOOL;	(*应急泵*)



	left_side_choice 										: BOOL;	(*左单边*)
	right_side_choice										: BOOL;	(*右单边*)

	level_extend_triger_left								: BOOL;	(*自动伸支腿*)
	level_extend_triger_right								: BOOL;	(*自动伸支腿*)
	auto_extend_triger_left								: BOOL;	(*自动伸支腿*)
	auto_extend_triger_right								: BOOL;	(*自动伸支腿*)
	auto_drawback_triger_left							: BOOL;	(*自动收支腿*)
	auto_drawback_triger_right							: BOOL;	(*自动收支腿*)

	level_extend_triger_left1		AT %IX34.2			: BOOL;	(*自动伸支腿*)
	level_extend_triger_right1	AT %IX34.3			: BOOL;	(*自动伸支腿*)
	auto_extend_triger_left1		AT %IX33.5			: BOOL;	(*自动伸支腿*)
	auto_extend_triger_right1	AT %IX33.6			: BOOL;	(*自动伸支腿*)
	auto_drawback_triger_left1	AT %IX33.7			: BOOL;	(*自动收支腿*)
	auto_drawback_triger_right1	AT %IX34.0			: BOOL;	(*自动收支腿*)


(***检测***)
	arm_to_station				AT %IX2.4				: BOOL;	(*臂架到位检测*)
	water_pump_check			AT %IX33.4			: BOOL;	(*水泵取力*)
	left_groud_check1			AT %IX34.4			: BOOL;	(*车胎离地1*)
	left_groud_check2			AT %IX34.5			: BOOL;	(*车胎离地2*)
	oil_pump_check										: BOOL;	(*油泵检测*)

(***支腿遥控盒***)
	remote_switch_leg									: BOOL;	(*支腿选择*)
	remote_control_left									: BOOL;	(*支腿左*)
	remote_control_right									: BOOL;	(*支腿右*)
	remote_control_up									: BOOL;	(*支腿上*)
	remote_control_down								: BOOL;	(*支腿下*)
	remote_out_front_left									: BOOL;	(*指示灯左前*)
	remote_out_front_back								: BOOL;	(*指示灯左后*)
	remote_out_right_left									: BOOL;	(*指示灯右前*)
	remote_out_right_back								: BOOL;	(*指示灯右后*)

(*************************************D_OUTPUT*****************************************)
(***支腿***)
	left_front_lv_ex_valve			AT %QX32.2	 		:  BOOL;	(*左前水平伸*)
	left_back_lv_ex_valve			AT %QX32.0 			:  BOOL;	(*左后水平伸*)
	right_front_lv_ex_valve		AT %QX32.6			:  BOOL;	(*右前水平伸*)
	right_back_lv_ex_valve		AT %QX32.4			:  BOOL;	(*右后水平伸*)
	left_front_lv_drb_valve		AT %QX32.3	 		:  BOOL;	(*左前水平收*)
	left_back_lv_drb_valve		AT %QX32.1 			:  BOOL;	(*左后水平收*)
	right_front_lv_drb_valve		AT %QX32.7			:  BOOL;	(*右前水平收*)
	right_back_lv_drb_valve		AT %QX32.5			:  BOOL;	(*右后水平收*)

(***底盘***)
	enginer_run_ctl				AT %QX0.8	 		:  BOOL;	(*启动控制*)
	enginer_stop_ctl				AT %QX0.9	 		:  BOOL;	(*熄火控制*)
	enginer_acc_ctl				AT %QX32.9	 		:  BOOL;	(*加速控制*)
	enginer_dec_ctl				AT %QX32.10	 		:  BOOL;	(*减速控制*)

(***操作***)
	water_pump_ctl				AT %QX0.10	 		:  BOOL;	(*水泵控制*)
	standby_oil_pump							 		:  BOOL;	(*应急泵*)
	up_valve_ctl					AT %QX32.14	 		:  BOOL;	(*上车阀*)
	down_valve_ctl				AT %QX32.15 			:  BOOL;	(*下车阀*)

(***指示***)
	over_level_sign				AT %QX0.11	 		:  BOOL;	(*坡度超限*)
	triger_left_grd_sign			AT %QX0.12	 		:  BOOL;	(*支腿离地*)
	alarmer_horn					AT %QX32.8	 		:  BOOL;	(*警报器*)
	triger_flash					AT %QX32.13	 		:  BOOL;	(*支腿闪光灯*)
	triger_no_drawback_sign					 		:  BOOL;	(*支腿未全缩指示*)
	leveled_sign											:  BOOL;	(*下车调平指示*)
	water_pump_ctl_sign			AT %QX0.10	 		:  BOOL;	(*水泵控制指示*)

	canon_valve_open 			 (*AT %QX32.11*)		:  BOOL;(*消防炮气阀检测25E*)
	canon_valve_close			(* AT %QX32.12*)		:  BOOL;(*消防炮气阀检测25E*)

	left_f_lv_ex_over				AT %QX0.14	 		:  BOOL;	(*左前水平伸到位*)
	left_b_lv_ex_over				AT %QX0.15	 		:  BOOL;	(*左后水平伸到位*)
	right_f_lv_ex_over				AT %QX32.11	 		:  BOOL;	(*右前水平伸到位*)
	right_b_lv_ex_over			AT %QX32.12	 		:  BOOL;	(*右后水平伸到位*)
	up_work_sign											:  BOOL;	(*上车工作指示*)
	down_work_sign										:  BOOL;	(*下车工作指示*)
	under_reset_ctl								 		:  BOOL;	(*底盘复位*)

END_VAR

(* Global variable list: VEHICLE TYPE/io_Variables_10012 *)
VAR_GLOBAL
(*************************************A_INPUT*******************************************)
	angle_x												: INT;		(*倾角X轴*)
	angle_y												: INT;		(*倾角Y轴*)
	angle_x_1												: INT;
	angle_y_1												: INT;
	oil_pressure											: WORD;	(*油压*)
	water_pressure										: WORD;	(*系统水压*)
	water_height_sign									: WORD;	(*水位信号*)
	foam_height_sign									: WORD;	(*泡沫液位信号*)
	water_flux												: WORD;	(*水流量信号*)
	speed_sign											: WORD;	(*速度脉冲*)

(**************************************A_OUTPUT***************************************)
	left_front_desired										: WORD;	(*左前垂直伸*)
	right_front_desired									: WORD;	(*右前垂直伸*)
	left_back_desired										: WORD;	(*左后垂直伸*)
	right_back_desired									: WORD;	(*右后垂直伸*)

	right_front_drawback_desired						: WORD;	(*右前垂直收*)
	left_back_drawback_desired							: WORD;	(*左后垂直收*)
	right_back_drawback_desired						: WORD;	(*右后垂直收*)
	left_front_drawback_desired							: WORD;	(*左前垂直收*)

(*************************************D_INPUT*******************************************)
(***支腿***)
	front_left_Lv_ex_check1		AT %IX0.6				: BOOL;	(*左前水平伸到位*)
	front_right_Lv_ex_check1		AT %IX0.7				: BOOL;	(*右前水平伸到位*)
	back_left_Lv_ex_check1		AT %IX0.12			: BOOL;	(*左后水平伸到位*)
	back_right_Lv_ex_check1	AT %IX0.13			: BOOL;	(*右后水平伸到位*)
	front_left_urt_ex_check1		AT %IX0.14			: BOOL;	(*左前垂直伸到位*)
	front_right_urt_ex_check1	AT %IX0.15			: BOOL;	(*右前垂直伸到位*)
	back_left_urt_ex_check1		AT %IX1.4				: BOOL;	(*左后垂直伸到位*)
	back_right_urt_ex_check1	AT %IX1.5				: BOOL;	(*右后垂直伸到位*)

	front_left_Lv_ex_check								: BOOL;	(*左前水平伸到位*)
	front_right_Lv_ex_check								: BOOL;	(*右前水平伸到位*)
	back_left_Lv_ex_check								: BOOL;	(*左后水平伸到位*)
	back_right_Lv_ex_check								: BOOL;	(*右后水平伸到位*)
	front_left_urt_ex_check								: BOOL;	(*左前垂直伸到位*)
	front_right_urt_ex_check								: BOOL;	(*右前垂直伸到位*)
	back_left_urt_ex_check								: BOOL;	(*左后垂直伸到位*)
	back_right_urt_ex_check								: BOOL;	(*右后垂直伸到位*)

	front_left_Lv_drb_check		AT %IX32.1			: BOOL;	(*左前水平收到位*)
	front_right_Lv_drb_check		AT %IX32.2			: BOOL;	(*右前水平收到位*)
	back_left_Lv_drb_check		AT %IX32.3			: BOOL;	(*左后水平收到位*)
	back_right_Lv_drb_check	AT %IX32.4			: BOOL;	(*右后水平收到位*)
	front_left_urt_drb_check1		AT %IX32.5			: BOOL;	(*左前垂直收到位*)
	front_right_urt_drb_check1	AT %IX32.6			: BOOL;	(*右前垂直收到位*)
	back_left_urt_drb_check1	AT %IX32.7			: BOOL;	(*左后垂直收到位*)
	back_right_urt_drb_check1	AT %IX32.12			: BOOL;	(*右后垂直收到位*)

	front_left_urt_drb_check								: BOOL;	(*左前垂直收到位*)
	front_right_urt_drb_check							: BOOL;	(*右前垂直收到位*)
	back_left_urt_drb_check								: BOOL;	(*左后垂直收到位*)
	back_right_urt_drb_check							: BOOL;	(*右后垂直收到位*)

(***底盘***)
	engine_run					AT %IX2.2				: BOOL;	(*发动机启动*)
	engine_stop					AT %IX2.3				: BOOL;	(*发动机停止*)
	accelerate_sb					AT %IX2.0				: BOOL;	(*加速*)
	decelerate_sb					AT %IX2.1				: BOOL;	(*减速*)

(***操作***)
	tt_forcexx						AT %IX34.6			: BOOL;	(*转台强制*)
	down_force					AT %IX34.7			: BOOL;	(*下车强制*)
	auto_manu_choice			AT %IX34.1			: BOOL;	(*自动/手动*)
	water_pump_run_sb			AT %IX1.7				: BOOL;	(*消防泵开*)
	standby_pump_check								: BOOL;	(*应急泵*)



	left_side_choice 										: BOOL;	(*左单边*)
	right_side_choice										: BOOL;	(*右单边*)

	level_extend_triger_left								: BOOL;	(*自动伸支腿*)
	level_extend_triger_right								: BOOL;	(*自动伸支腿*)
	auto_extend_triger_left								: BOOL;	(*自动伸支腿*)
	auto_extend_triger_right								: BOOL;	(*自动伸支腿*)
	auto_drawback_triger_left							: BOOL;	(*自动收支腿*)
	auto_drawback_triger_right							: BOOL;	(*自动收支腿*)

	level_extend_triger_left1		(*AT %IX34.2*)		: BOOL;	(*自动伸支腿*)
	level_extend_triger_right1	(*AT %IX34.3*)		: BOOL;	(*自动伸支腿*)
	auto_extend_triger_left1		(*AT %IX33.5*)		: BOOL;	(*自动伸支腿*)
	auto_extend_triger_right1	(*AT %IX33.6*)		: BOOL;	(*自动伸支腿*)
	auto_drawback_triger_left1	(*AT %IX33.7*)		: BOOL;	(*自动收支腿*)
	auto_drawback_triger_right1	(*AT %IX34.0*)		: BOOL;	(*自动收支腿*)


(***检测***)
	arm_to_station				AT %IX2.4				: BOOL;	(*臂架到位检测*)
	water_pump_check			AT %IX33.4			: BOOL;	(*水泵取力*)
	left_groud_check1			AT %IX34.4			: BOOL;	(*车胎离地1*)
	left_groud_check2			AT %IX34.5			: BOOL;	(*车胎离地2*)
	oil_pump_check				AT %IX32.15			: BOOL;	(*油泵检测*)

(***支腿遥控盒***)
	remote_switch_leg									: BOOL;	(*支腿选择*)
	remote_control_left									: BOOL;	(*支腿左*)
	remote_control_right									: BOOL;	(*支腿右*)
	remote_control_up									: BOOL;	(*支腿上*)
	remote_control_down								: BOOL;	(*支腿下*)
	remote_out_front_left									: BOOL;	(*指示灯左前*)
	remote_out_front_back								: BOOL;	(*指示灯左后*)
	remote_out_right_left									: BOOL;	(*指示灯右前*)
	remote_out_right_back								: BOOL;	(*指示灯右后*)

(*************************************D_OUTPUT*****************************************)
(***支腿***)
	left_front_lv_ex_valve			AT %QX32.2	 		:  BOOL;	(*左前水平伸*)
	left_back_lv_ex_valve			AT %QX32.0 			:  BOOL;	(*左后水平伸*)
	right_front_lv_ex_valve		AT %QX32.6			:  BOOL;	(*右前水平伸*)
	right_back_lv_ex_valve		AT %QX32.4			:  BOOL;	(*右后水平伸*)
	left_front_lv_drb_valve		AT %QX32.3	 		:  BOOL;	(*左前水平收*)
	left_back_lv_drb_valve		AT %QX32.1 			:  BOOL;	(*左后水平收*)
	right_front_lv_drb_valve		AT %QX32.7			:  BOOL;	(*右前水平收*)
	right_back_lv_drb_valve		AT %QX32.5			:  BOOL;	(*右后水平收*)

(***底盘***)
	enginer_run_ctl				AT %QX0.8	 		:  BOOL;	(*启动控制*)
	enginer_stop_ctl				AT %QX0.9	 		:  BOOL;	(*熄火控制*)
	enginer_acc_ctl				AT %QX32.9	 		:  BOOL;	(*加速控制*)
	enginer_dec_ctl				AT %QX32.10	 		:  BOOL;	(*减速控制*)

(***操作***)
	water_pump_ctl				AT %QX0.10	 		:  BOOL;	(*水泵控制*)
	standby_oil_pump							 		:  BOOL;	(*应急泵*)
	up_valve_ctl					AT %QX32.14	 		:  BOOL;	(*上车阀*)
	down_valve_ctl				AT %QX32.15 			:  BOOL;	(*下车阀*)

(***指示***)
	over_level_sign				AT %QX0.11	 		:  BOOL;	(*坡度超限*)
	triger_left_grd_sign			AT %QX0.12	 		:  BOOL;	(*支腿离地*)
	alarmer_horn					AT %QX32.8	 		:  BOOL;	(*警报器*)
	triger_flash					AT %QX32.13	 		:  BOOL;	(*支腿闪光灯*)
	triger_no_drawback_sign	AT %QX0.15	 		:  BOOL;	(*支腿未全缩指示*)
	leveled_sign					AT %QX0.14			:  BOOL;	(*下车调平指示*)
	water_pump_ctl_sign			AT %QX0.10	 		:  BOOL;	(*水泵控制指示*)

	canon_valve_open 			 (*AT %QX32.11*)		:  BOOL;(*消防炮气阀检测25E*)
	canon_valve_close			(* AT %QX32.12*)		:  BOOL;(*消防炮气阀检测25E*)

	left_f_lv_ex_over				(*AT %QX0.14*)	 	:  BOOL;	(*左前水平伸到位*)
	left_b_lv_ex_over				(*AT %QX0.15*) 		:  BOOL;	(*左后水平伸到位*)
	right_f_lv_ex_over				(*AT %QX32.11*)	 	:  BOOL;	(*右前水平伸到位*)
	right_b_lv_ex_over			(*AT %QX32.12*) 		:  BOOL;	(*右后水平伸到位*)
	up_work_sign											:  BOOL;	(*上车工作指示*)
	down_work_sign										:  BOOL;	(*下车工作指示*)
	under_reset_ctl								 		:  BOOL;	(*底盘复位*)

END_VAR

(* Global variable list: VEHICLE TYPE/io_Variables_10013 *)
VAR_GLOBAL
(*************************************A_INPUT*******************************************)
	angle_x												: INT;		(*倾角X轴*)
	angle_y												: INT;		(*倾角Y轴*)
	angle_x_1												: INT;
	angle_y_1												: INT;
	oil_pressure											: WORD;	(*油压*)
	water_pressure										: WORD;	(*系统水压*)
	water_height_sign									: WORD;	(*水位信号*)
	foam_height_sign									: WORD;	(*泡沫液位信号*)
	water_flux												: WORD;	(*水流量信号*)
	speed_sign											: WORD;	(*速度脉冲*)

(**************************************A_OUTPUT***************************************)
	left_front_desired										: WORD;	(*左前垂直伸*)
	right_front_desired									: WORD;	(*右前垂直伸*)
	left_back_desired										: WORD;	(*左后垂直伸*)
	right_back_desired									: WORD;	(*右后垂直伸*)

	right_front_drawback_desired						: WORD;	(*右前垂直收*)
	left_back_drawback_desired							: WORD;	(*左后垂直收*)
	right_back_drawback_desired						: WORD;	(*右后垂直收*)
	left_front_drawback_desired							: WORD;	(*左前垂直收*)

(*************************************D_INPUT*******************************************)
(***支腿***)
	front_left_Lv_ex_check1		AT %IX0.6				: BOOL;	(*左前水平伸到位*)
	front_right_Lv_ex_check1		AT %IX0.7				: BOOL;	(*右前水平伸到位*)
	back_left_Lv_ex_check1		AT %IX0.12			: BOOL;	(*左后水平伸到位*)
	back_right_Lv_ex_check1	AT %IX0.13			: BOOL;	(*右后水平伸到位*)
	front_left_urt_ex_check1		AT %IX0.14			: BOOL;	(*左前垂直伸到位*)
	front_right_urt_ex_check1	AT %IX0.15			: BOOL;	(*右前垂直伸到位*)
	back_left_urt_ex_check1		AT %IX1.4				: BOOL;	(*左后垂直伸到位*)
	back_right_urt_ex_check1	AT %IX1.5				: BOOL;	(*右后垂直伸到位*)

	front_left_Lv_ex_check								: BOOL;	(*左前水平伸到位*)
	front_right_Lv_ex_check								: BOOL;	(*右前水平伸到位*)
	back_left_Lv_ex_check								: BOOL;	(*左后水平伸到位*)
	back_right_Lv_ex_check								: BOOL;	(*右后水平伸到位*)
	front_left_urt_ex_check								: BOOL;	(*左前垂直伸到位*)
	front_right_urt_ex_check								: BOOL;	(*右前垂直伸到位*)
	back_left_urt_ex_check								: BOOL;	(*左后垂直伸到位*)
	back_right_urt_ex_check								: BOOL;	(*右后垂直伸到位*)

	front_left_Lv_drb_check		AT %IX32.1			: BOOL;	(*左前水平收到位*)
	front_right_Lv_drb_check		AT %IX32.2			: BOOL;	(*右前水平收到位*)
	back_left_Lv_drb_check		AT %IX32.3			: BOOL;	(*左后水平收到位*)
	back_right_Lv_drb_check	AT %IX32.4			: BOOL;	(*右后水平收到位*)
	front_left_urt_drb_check1		AT %IX32.5			: BOOL;	(*左前垂直收到位*)
	front_right_urt_drb_check1	AT %IX32.6			: BOOL;	(*右前垂直收到位*)
	back_left_urt_drb_check1	AT %IX32.7			: BOOL;	(*左后垂直收到位*)
	back_right_urt_drb_check1	AT %IX32.12			: BOOL;	(*右后垂直收到位*)

	front_left_urt_drb_check								: BOOL;	(*左前垂直收到位*)
	front_right_urt_drb_check							: BOOL;	(*右前垂直收到位*)
	back_left_urt_drb_check								: BOOL;	(*左后垂直收到位*)
	back_right_urt_drb_check							: BOOL;	(*右后垂直收到位*)

(***底盘***)
	engine_run					AT %IX2.2				: BOOL;	(*发动机启动*)
	engine_stop					AT %IX2.3				: BOOL;	(*发动机停止*)
	accelerate_sb					AT %IX2.0				: BOOL;	(*加速*)
	decelerate_sb					AT %IX2.1				: BOOL;	(*减速*)

(***操作***)
	tt_forcexx						AT %IX34.6			: BOOL;	(*转台强制*)
	down_force					AT %IX34.7			: BOOL;	(*下车强制*)
	auto_manu_choice			AT %IX34.1			: BOOL;	(*自动/手动*)
	water_pump_run_sb			AT %IX1.7				: BOOL;	(*消防泵开*)
	standby_pump_check								: BOOL;	(*应急泵*)



	left_side_choice 										: BOOL;	(*左单边*)
	right_side_choice										: BOOL;	(*右单边*)

	level_extend_triger_left								: BOOL;	(*自动伸支腿*)
	level_extend_triger_right								: BOOL;	(*自动伸支腿*)
	auto_extend_triger_left								: BOOL;	(*自动伸支腿*)
	auto_extend_triger_right								: BOOL;	(*自动伸支腿*)
	auto_drawback_triger_left							: BOOL;	(*自动收支腿*)
	auto_drawback_triger_right							: BOOL;	(*自动收支腿*)

	level_extend_triger_left1		(*AT %IX34.2*)		: BOOL;	(*自动伸支腿*)
	level_extend_triger_right1	(*AT %IX34.3*)		: BOOL;	(*自动伸支腿*)
	auto_extend_triger_left1		(*AT %IX33.5*)		: BOOL;	(*自动伸支腿*)
	auto_extend_triger_right1	(*AT %IX33.6*)		: BOOL;	(*自动伸支腿*)
	auto_drawback_triger_left1	(*AT %IX33.7*)		: BOOL;	(*自动收支腿*)
	auto_drawback_triger_right1	(*AT %IX34.0*)		: BOOL;	(*自动收支腿*)


(***检测***)
	arm_to_station				AT %IX2.4				: BOOL;	(*臂架到位检测*)
	water_pump_check			AT %IX33.4			: BOOL;	(*水泵取力*)
	left_groud_check1			AT %IX34.4			: BOOL;	(*车胎离地1*)
	left_groud_check2			AT %IX34.5			: BOOL;	(*车胎离地2*)
	oil_pump_check										: BOOL;	(*油泵检测*)

(***支腿遥控盒***)
	remote_switch_leg									: BOOL;	(*支腿选择*)
	remote_control_left									: BOOL;	(*支腿左*)
	remote_control_right									: BOOL;	(*支腿右*)
	remote_control_up									: BOOL;	(*支腿上*)
	remote_control_down								: BOOL;	(*支腿下*)
	remote_out_front_left									: BOOL;	(*指示灯左前*)
	remote_out_front_back								: BOOL;	(*指示灯左后*)
	remote_out_right_left									: BOOL;	(*指示灯右前*)
	remote_out_right_back								: BOOL;	(*指示灯右后*)

(*************************************D_OUTPUT*****************************************)
(***支腿***)
	left_front_lv_ex_valve			AT %QX32.2	 		:  BOOL;	(*左前水平伸*)
	left_back_lv_ex_valve			AT %QX32.0 			:  BOOL;	(*左后水平伸*)
	right_front_lv_ex_valve		AT %QX32.6			:  BOOL;	(*右前水平伸*)
	right_back_lv_ex_valve		AT %QX32.4			:  BOOL;	(*右后水平伸*)
	left_front_lv_drb_valve		AT %QX32.3	 		:  BOOL;	(*左前水平收*)
	left_back_lv_drb_valve		AT %QX32.1 			:  BOOL;	(*左后水平收*)
	right_front_lv_drb_valve		AT %QX32.7			:  BOOL;	(*右前水平收*)
	right_back_lv_drb_valve		AT %QX32.5			:  BOOL;	(*右后水平收*)

(***底盘***)
	enginer_run_ctl				AT %QX0.8	 		:  BOOL;	(*启动控制*)
	enginer_stop_ctl				AT %QX0.9	 		:  BOOL;	(*熄火控制*)
	enginer_acc_ctl				AT %QX32.9	 		:  BOOL;	(*加速控制*)
	enginer_dec_ctl				AT %QX32.10	 		:  BOOL;	(*减速控制*)

(***操作***)
	water_pump_ctl				AT %QX0.10	 		:  BOOL;	(*水泵控制*)
	standby_oil_pump							 		:  BOOL;	(*应急泵*)
	up_valve_ctl					AT %QX32.14	 		:  BOOL;	(*上车阀*)
	down_valve_ctl				AT %QX32.15 			:  BOOL;	(*下车阀*)

(***指示***)
	over_level_sign				AT %QX0.11	 		:  BOOL;	(*坡度超限*)
	triger_left_grd_sign			AT %QX0.12	 		:  BOOL;	(*支腿离地*)
	alarmer_horn					AT %QX32.8	 		:  BOOL;	(*警报器*)
	triger_flash					AT %QX32.13	 		:  BOOL;	(*支腿闪光灯*)
	triger_no_drawback_sign	AT %QX0.15	 		:  BOOL;	(*支腿未全缩指示*)
	leveled_sign					AT %QX0.14	 		:  BOOL;	(*下车调平指示*)
	water_pump_ctl_sign			AT %QX0.10	 		:  BOOL;	(*水泵控制指示*)

	canon_valve_open 			 (*AT %QX32.11*)		:  BOOL;(*消防炮气阀检测25E*)
	canon_valve_close			(* AT %QX32.12*)		:  BOOL;(*消防炮气阀检测25E*)

	left_f_lv_ex_over								 		:  BOOL;	(*左前水平伸到位*)
	left_b_lv_ex_over								 		:  BOOL;	(*左后水平伸到位*)
	right_f_lv_ex_over								 		:  BOOL;	(*右前水平伸到位*)
	right_b_lv_ex_over							 		:  BOOL;	(*右后水平伸到位*)
	up_work_sign											:  BOOL;	(*上车工作指示*)
	down_work_sign										:  BOOL;	(*下车工作指示*)
	under_reset_ctl								 		:  BOOL;	(*底盘复位*)

END_VAR

(* Global variable list: VEHICLE TYPE/io_Variables_10014 *)
VAR_GLOBAL
(*************************************A_INPUT*******************************************)
	angle_x												: INT;		(*倾角X轴*)
	angle_y												: INT;		(*倾角Y轴*)
	angle_x_1												: INT;
	angle_y_1												: INT;
	oil_pressure											: WORD;	(*油压*)
	water_pressure										: WORD;	(*系统水压*)
	water_height_sign									: WORD;	(*水位信号*)
	foam_height_sign									: WORD;	(*泡沫液位信号*)
	water_flux												: WORD;	(*水流量信号*)
	speed_sign											: WORD;	(*速度脉冲*)

(**************************************A_OUTPUT***************************************)
	left_front_desired										: WORD;	(*左前垂直伸*)
	right_front_desired									: WORD;	(*右前垂直伸*)
	left_back_desired										: WORD;	(*左后垂直伸*)
	right_back_desired									: WORD;	(*右后垂直伸*)

	right_front_drawback_desired						: WORD;	(*右前垂直收*)
	left_back_drawback_desired							: WORD;	(*左后垂直收*)
	right_back_drawback_desired						: WORD;	(*右后垂直收*)
	left_front_drawback_desired							: WORD;	(*左前垂直收*)

(*************************************D_INPUT*******************************************)
(***支腿***)
	front_left_Lv_ex_check1		AT %IX0.6				: BOOL;	(*左前水平伸到位*)
	front_right_Lv_ex_check1		AT %IX0.7				: BOOL;	(*右前水平伸到位*)
	back_left_Lv_ex_check1		AT %IX0.12			: BOOL;	(*左后水平伸到位*)
	back_right_Lv_ex_check1	AT %IX0.13			: BOOL;	(*右后水平伸到位*)
	front_left_urt_ex_check1		AT %IX0.14			: BOOL;	(*左前垂直伸到位*)
	front_right_urt_ex_check1	AT %IX0.15			: BOOL;	(*右前垂直伸到位*)
	back_left_urt_ex_check1		AT %IX1.4				: BOOL;	(*左后垂直伸到位*)
	back_right_urt_ex_check1	AT %IX1.5				: BOOL;	(*右后垂直伸到位*)

	front_left_Lv_ex_check								: BOOL;	(*左前水平伸到位*)
	front_right_Lv_ex_check								: BOOL;	(*右前水平伸到位*)
	back_left_Lv_ex_check								: BOOL;	(*左后水平伸到位*)
	back_right_Lv_ex_check								: BOOL;	(*右后水平伸到位*)
	front_left_urt_ex_check								: BOOL;	(*左前垂直伸到位*)
	front_right_urt_ex_check								: BOOL;	(*右前垂直伸到位*)
	back_left_urt_ex_check								: BOOL;	(*左后垂直伸到位*)
	back_right_urt_ex_check								: BOOL;	(*右后垂直伸到位*)

	front_left_Lv_drb_check		AT %IX32.1			: BOOL;	(*左前水平收到位*)
	front_right_Lv_drb_check		AT %IX32.2			: BOOL;	(*右前水平收到位*)
	back_left_Lv_drb_check		AT %IX32.3			: BOOL;	(*左后水平收到位*)
	back_right_Lv_drb_check	AT %IX32.4			: BOOL;	(*右后水平收到位*)
	front_left_urt_drb_check1		AT %IX32.5			: BOOL;	(*左前垂直收到位*)
	front_right_urt_drb_check1	AT %IX32.6			: BOOL;	(*右前垂直收到位*)
	back_left_urt_drb_check1	AT %IX32.7			: BOOL;	(*左后垂直收到位*)
	back_right_urt_drb_check1	AT %IX32.12			: BOOL;	(*右后垂直收到位*)

	front_left_urt_drb_check								: BOOL;	(*左前垂直收到位*)
	front_right_urt_drb_check							: BOOL;	(*右前垂直收到位*)
	back_left_urt_drb_check								: BOOL;	(*左后垂直收到位*)
	back_right_urt_drb_check							: BOOL;	(*右后垂直收到位*)

(***底盘***)
	engine_run					AT %IX1.10			: BOOL;	(*发动机启动*)
	engine_stop					AT %IX1.11			: BOOL;	(*发动机停止*)
	accelerate_sb					AT %IX1.8				: BOOL;	(*加速*)
	decelerate_sb					AT %IX1.9				: BOOL;	(*减速*)

(***操作***)
	tt_forcexx						AT %IX33.14			: BOOL;	(*转台强制*)
	down_force					AT %IX33.15			: BOOL;	(*下车强制*)
	auto_manu_choice			AT %IX33.5			: BOOL;	(*自动/手动*)
	water_pump_run_sb			AT %IX1.7				: BOOL;	(*消防泵开*)
	standby_pump_check								: BOOL;	(*应急泵*)



	left_side_choice 										: BOOL;	(*左单边*)
	right_side_choice										: BOOL;	(*右单边*)

	level_extend_triger_left								: BOOL;	(*自动伸支腿*)
	level_extend_triger_right								: BOOL;	(*自动伸支腿*)
	auto_extend_triger_left								: BOOL;	(*自动伸支腿*)
	auto_extend_triger_right								: BOOL;	(*自动伸支腿*)
	auto_drawback_triger_left							: BOOL;	(*自动收支腿*)
	auto_drawback_triger_right							: BOOL;	(*自动收支腿*)

	level_extend_triger_left1		(*AT %IX34.2*)		: BOOL;	(*自动伸支腿*)
	level_extend_triger_right1	(*AT %IX34.3*)		: BOOL;	(*自动伸支腿*)
	auto_extend_triger_left1		(*AT %IX33.5*)		: BOOL;	(*自动伸支腿*)
	auto_extend_triger_right1	(*AT %IX33.6*)		: BOOL;	(*自动伸支腿*)
	auto_drawback_triger_left1	(*AT %IX33.7*)		: BOOL;	(*自动收支腿*)
	auto_drawback_triger_right1	(*AT %IX34.0*)		: BOOL;	(*自动收支腿*)


(***检测***)
	arm_to_station				AT %IX1.12			: BOOL;	(*臂架到位检测*)
	water_pump_check			(*AT %IX33.4*)		: BOOL;	(*水泵取力*)
	left_groud_check1			AT %IX33.12			: BOOL;	(*车胎离地1*)
	left_groud_check2			AT %IX33.13			: BOOL;	(*车胎离地2*)
	oil_pump_check										: BOOL;	(*油泵检测*)

(***支腿遥控盒***)
	remote_switch_leg									: BOOL;	(*支腿选择*)
	remote_control_left									: BOOL;	(*支腿左*)
	remote_control_right									: BOOL;	(*支腿右*)
	remote_control_up									: BOOL;	(*支腿上*)
	remote_control_down								: BOOL;	(*支腿下*)
	remote_out_front_left									: BOOL;	(*指示灯左前*)
	remote_out_front_back								: BOOL;	(*指示灯左后*)
	remote_out_right_left									: BOOL;	(*指示灯右前*)
	remote_out_right_back								: BOOL;	(*指示灯右后*)

(*************************************D_OUTPUT*****************************************)
(***支腿***)
	left_front_lv_ex_valve			AT %QX32.2	 		:  BOOL;	(*左前水平伸*)
	left_back_lv_ex_valve			AT %QX32.0 			:  BOOL;	(*左后水平伸*)
	right_front_lv_ex_valve		AT %QX32.6			:  BOOL;	(*右前水平伸*)
	right_back_lv_ex_valve		AT %QX32.4			:  BOOL;	(*右后水平伸*)
	left_front_lv_drb_valve		AT %QX32.3	 		:  BOOL;	(*左前水平收*)
	left_back_lv_drb_valve		AT %QX32.1 			:  BOOL;	(*左后水平收*)
	right_front_lv_drb_valve		AT %QX32.7			:  BOOL;	(*右前水平收*)
	right_back_lv_drb_valve		AT %QX32.5			:  BOOL;	(*右后水平收*)

(***底盘***)
	enginer_run_ctl				AT %QX1.0	 		:  BOOL;	(*启动控制*)
	enginer_stop_ctl				AT %QX1.1	 		:  BOOL;	(*熄火控制*)
	enginer_acc_ctl				AT %QX33.1	 		:  BOOL;	(*加速控制*)
	enginer_dec_ctl				AT %QX33.2	 		:  BOOL;	(*减速控制*)

(***操作***)
	water_pump_ctl				AT %QX1.2	 		:  BOOL;	(*水泵控制*)
	standby_oil_pump							 		:  BOOL;	(*应急泵*)
	up_valve_ctl					AT %QX33.6	 		:  BOOL;	(*上车阀*)
	down_valve_ctl				AT %QX33.7 			:  BOOL;	(*下车阀*)

(***指示***)
	over_level_sign				AT %QX1.3		 	:  BOOL;	(*坡度超限*)
	triger_left_grd_sign			AT %QX1.4		 	:  BOOL;	(*支腿离地*)
	alarmer_horn					AT %QX33.0		 	:  BOOL;	(*警报器*)
	triger_flash					AT %QX33.5		 	:  BOOL;	(*支腿闪光灯*)
	triger_no_drawback_sign	AT %QX1.6		 	:  BOOL;	(*支腿未全缩指示*)
	leveled_sign					AT %QX1.5		 	:  BOOL;	(*下车调平指示*)
	water_pump_ctl_sign			(*AT %QX0.10*)	 	:  BOOL;	(*水泵控制指示*)

	canon_valve_open 			 (*AT %QX32.11*)		:  BOOL;(*消防炮气阀检测25E*)
	canon_valve_close			(* AT %QX32.12*)		:  BOOL;(*消防炮气阀检测25E*)

	left_f_lv_ex_over								 		:  BOOL;	(*左前水平伸到位*)
	left_b_lv_ex_over								 		:  BOOL;	(*左后水平伸到位*)
	right_f_lv_ex_over								 		:  BOOL;	(*右前水平伸到位*)
	right_b_lv_ex_over							 		:  BOOL;	(*右后水平伸到位*)
	up_work_sign											:  BOOL;	(*上车工作指示*)
	down_work_sign										:  BOOL;	(*下车工作指示*)
	under_reset_ctl								 		:  BOOL;	(*底盘复位*)

END_VAR

(* Global variable list: leg_test *)
VAR_GLOBAL RETAIN

END_VAR

VAR_GLOBAL

	leg_test						:BOOL;
	leg_test_m					:BOOL;

	ll_f:ARRAY[0..10] OF POINT       :=(X:=0,Y:=504),(X:=100,Y:=463),  (X:=200,Y:=421), (X:=300,Y:=380), 	(X:=400,Y:=339), 	(X:=500,Y:=298), 	(X:=600,Y:=257), 4((X:=1000,Y:=200));
	ll_b:ARRAY[0..10] OF POINT      :=(X:=0,Y:=504),(X:=100,Y:=534),  (X:=200,Y:=564), (X:=300,Y:=594), 	(X:=400,Y:=624), 	(X:=500,Y:=654), 	(X:=600,Y:=684), 4((X:=1000,Y:=700));
END_VAR


VAR_GLOBAL RETAIN
	front_left_urt_time_W			:WORD;
	front_right_urt_time_W		:WORD;
	back_left_urt_time_W			:WORD;
	back_right_urt_time_W		:WORD;
END_VAR

(* Global variable list: Networkmanagement implicit Variables CAN *)
VAR_GLOBAL CONSTANT
	USE_NWVARS_CAN : BOOL := TRUE;
	MAX_NetVarItems_CAN	: INT := 175;
	MAX_NetVarPDO_Rx_CAN	: INT := 10;
	MAX_NetVarPDO_Tx_CAN	: INT := 10;
	MAX_NetVarOD_CAN		: INT := 0;
END_VAR
VAR_GLOBAL
	pNetVarItems_CAN		: ARRAY[0..MAX_NetVarItems_CAN] OF NetVarDataItem_CAN;
	pNetVarPDO_Rx_CAN		: ARRAY[0..MAX_NetVarPDO_Rx_CAN] OF NetVarPDO_Rx_CAN;
	pNetVarPDO_Tx_CAN		: ARRAY[0..MAX_NetVarPDO_Tx_CAN] OF NetVarPDO_Tx_CAN;
	pNetVarOD_CAN			: ARRAY[0..MAX_NetVarOD_CAN] OF NetVarOD_CAN;
END_VAR

(* Global variable list: PDM_COMMUNICATION *)
VAR_GLOBAL
	(*
	Systemvariabelen f黵 die PLC-PDM Basiskommunikation. Bei CANopen: TX/RX PDO1 und PDO2 oder Layer2 TX/RX COB1 und COB2.
	Bei  CANopen mit EDS-File werden die Variabelen 黚er die AT - Adressierung zugewiesen. Entfernen Sie die Komentarzeichen f黵 die AT-Adresszuweisung
	und passen Sie die Adressen entsprechend Ihrer Steuerungskonfiguration an.

	Wenn Sie auf Basis Layer2 kommunizieren wollen, entfernen Sie nicht die Komentarzeichen. Kopieren Sie 黚er Projekt -> Kopieren... aus einem beliebigen Layer2-Template
	den Ordner PDM_COM_LAYER2.

	Ist die Steuerung als CANopen Slave konfiguriert m黶sen Sie ebenfalls auf Basis Layer2 mit dem dem PDM komunizieren. Aus diesem Grund beinhaltet
	ein PLC-Slave Template auch den Ordner PDM_COM_LAYER2.

	*************************************************************************************************************************************************************************************************

	System variables for the PLC-PDM basic communication. For CANopen: TX/RX PDO1 AND PDO2 or Layer2 TX/RX COB1 and COB2.
	For CANopen with EDS file the variables are assigned via the AT addressing. Remove the comment characters For the AT address assignment and adapt
	the addresses according to their control configuration.

	If you want to communicate on the Layer2 basis, do not remove the comment characters. Copy the folder PDM_COM_LAYER2 from any Layer2 template into
	your project via Project -> Merge...

	If the controller is configured as a CANopen slave, you also have to communicate with the PDM on the Layer2 basis. For this reason a PLC slave template
	also contains  the folder PDM_COM_LAYER2. If you do not need a PDM, you can simply delete this object and the folder PDN_COM_LAYER2 and the respective call in PLC_PRG.
	*)


	(*****************************variables from PLC to PDM******************************************)
	DESIRED_PAGE 					(*AT %QW32*)	: WORD;		(*Desired page number from PLC to PDM*)
	DESIRED_MESSAGE 			(*AT %QB66*)		: BYTE;			(*Desired message number from PLC to PDM*)
	DESIRED_MESSAGE_GROUP 	(*AT %QB67*)		:BYTE;			(*Desired message group number from PLC to PDM*)
	LED_F_KEYS 						(*AT %QB68*)		:BYTE;			(*LED Funtion keys from PLC to PDM*)
	LED_C_KEYS 					(*AT %QB69*)		:BYTE;			(*LED Control keys from PLC to PDM*)
	DESIRED_LEDVALUE_MAX 		(*AT %QB70*)		:BYTE;			(*Desired LED valus max from PLC to PDM*)
	DESIRED_LEDVALUE_NIGHT 	(*AT %QB71*)		:BYTE;			(*Desired LED value night from PLC to PDM*)
	DESIRED_BACKLIGHT 			(*AT %QB72*)		:BYTE;			(*Desired backlight value from PLC to PDM*)
	HANDLE_BACK 					(*AT %QW37*)	:WORD;		(*Handle for input value, write back from PLC to PDM*)
	INPUT_VALUE_BACK 			(*AT %QD19*)		:DWORD;		(*Input value, write back from PLC to PDM*)
	LENGHT_BACK 					(*AT %QB80*)		:BYTE;			(*Length for input value, write back from PLC to PDM*)

	(*****************************variables from PDM to PLC******************************************)
	PRESENT_PAGE 					(*AT %IW32*)		:WORD;		(*Present page number from PDM to PLC*)
	PRESENT_MESSAGE 			(*AT %IB66*)		:BYTE;			(*Present message number from PDM to PLC*)
	PRESENT_MESSAGE_GROUP	(*AT %IB67*)		:BYTE;			(*Present message group number from PDM to PLC*)
	F_KEYS 							(*AT %IB68*)		:BYTE;			(*Funtion keys from PDM to PLC*)
	C_KEYS 							(*AT %IB69*)		:BYTE;			(*Control keys from PDM to PLC*)
	PRESENT_LEDVALUE_MAX 		(*AT %IB70*)		:BYTE;			(*Present LED valus max from PDM to PLC*)
	PRESENT_LEDVALUE_NIGHT 	(*AT %IB71*)		:BYTE;			(*Present LED value night from PDM to PLC*)
	PRESENT_BACKLIGHT 			(*AT %IB72*)		:BYTE;			(*Present backlight value from PDM to PLC*)
	HANDLE				 			(*AT %IW37*)		:WORD;		(*Handle for input value from PDM to PLC*)
	INPUT_VALUE 					(*AT %ID19*)		:DWORD;		(*Input value from PDM to PLC*)
	LENGHT		 					(*AT %IB80*)		:BYTE;			(*Length for input value from PDM to PLC*)

END_VAR

(* Global variable list: var_cylinder_list *)
VAR_GLOBAL RETAIN

END_VAR

VAR_GLOBAL

	fl_o_fac_b: BOOL;
	fr_o_fac_b: BOOL;
	rl_o_fac_b: BOOL;
	rr_o_fac_b: BOOL;
	fl_i_fac_b: BOOL;
	fr_i_fac_b: BOOL;
	rl_i_fac_b: BOOL;
	rr_i_fac_b: BOOL;

	fl_o_fac_b_l: BOOL;
	fr_o_fac_b_l: BOOL;
	rl_o_fac_b_l: BOOL;
	rr_o_fac_b_l: BOOL;
	fl_i_fac_b_l: BOOL;
	fr_i_fac_b_l: BOOL;
	rl_i_fac_b_l: BOOL;
	rr_i_fac_b_l: BOOL;

	fl_o_fac_b_r: BOOL;
	fr_o_fac_b_r: BOOL;
	rl_o_fac_b_r: BOOL;
	rr_o_fac_b_r: BOOL;
	fl_i_fac_b_r: BOOL;
	fr_i_fac_b_r: BOOL;
	rl_i_fac_b_r: BOOL;
	rr_i_fac_b_r: BOOL;

	ramp_selected: BOOL;


	left_front_desired_CR0032										: WORD;(*左前垂直伸*)
	right_front_desired_CR0032									: WORD;(*右前垂直伸*)
	left_back_desired_CR0032										: WORD;(*左后垂直伸*)
	right_back_desired_CR0032									: WORD;(*右后垂直伸*)

END_VAR

VAR_GLOBAL
	fl_fac_nr 		AT%MW20:INT:=0;
	fl_fac_l_nr 	AT%MW22:INT:=0;
	fl_fac_r_nr 	AT%MW24:INT:=0;

	fr_fac_nr 		AT%MW26:INT:=0;
	fr_fac_l_nr 	AT%MW28:INT:=0;
	fr_fac_r_nr 	AT%MW30:INT:=0;

	rl_fac_nr 		AT%MW32:INT:=0;
	rl_fac_l_nr 	AT%MW34:INT:=0;
	rl_fac_r_nr 	AT%MW36:INT:=0;

	rr_fac_nr 		AT%MW38:INT:=0;
	rr_fac_l_nr 	AT%MW40:INT:=0;
	rr_fac_r_nr 	AT%MW42:INT:=0;

	fl_fac_nr2 		AT%MW44:INT:=0;
	fl_fac_l_nr2 	AT%MW46:INT:=0;
	fl_fac_r_nr2 	AT%MW48:INT:=0;

	fr_fac_nr2 		AT%MW50:INT:=0;
	fr_fac_l_nr2 	AT%MW52:INT:=0;
	fr_fac_r_nr2 	AT%MW54:INT:=0;

	rl_fac_nr2 		AT%MW56:INT:=0;
	rl_fac_l_nr2 	AT%MW58:INT:=0;
	rl_fac_r_nr2 	AT%MW60:INT:=0;

	rr_fac_nr2 		AT%MW62:INT:=0;
	rr_fac_l_nr2 	AT%MW64:INT:=0;
	rr_fac_r_nr2 	AT%MW66:INT:=0;
END_VAR

(* Data type *)
TYPE cc_point :
STRUCT
(*	a:INT;*)
	b:ARRAY[0..10] OF POINT ;
END_STRUCT
END_TYPE

(* POU PLC_PRG, FBD *)
PROGRAM PLC_PRG
VAR

	init_e: BOOL;
	cycletime: DWORD;
	max_cycletime: DWORD;
	reset_max:BOOL;


	ga: MEMORY_RETAIN_PARAM;
END_VAR
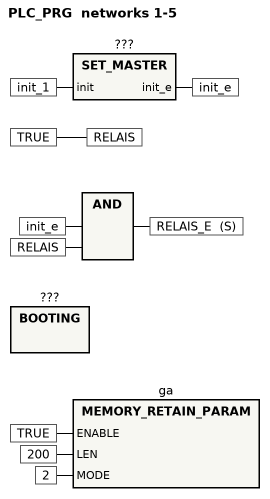
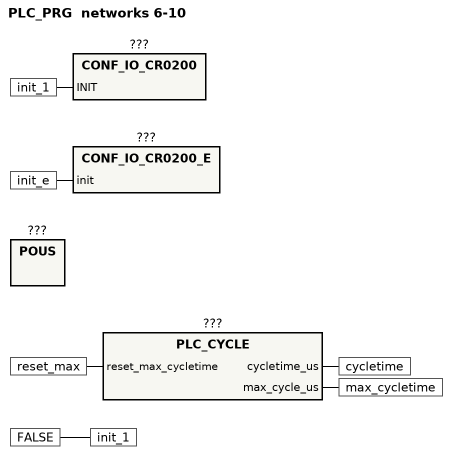
_FBD_ (* Function Block Diagram *)
NETWORK 1
	???:SET_MASTER(init: init_1) => init_e
NETWORK 2
	TRUE => RELAIS
NETWORK 3
	AND(init_e, RELAIS) => S RELAIS_E
NETWORK 4
	???:BOOTING()
NETWORK 5
	ga:MEMORY_RETAIN_PARAM(ENABLE: TRUE, LEN: 200, MODE: 2)
NETWORK 6
	???:CONF_IO_CR0200(INIT: init_1)
NETWORK 7
	???:CONF_IO_CR0200_E(init: init_e)
NETWORK 8
	???:POUS()
NETWORK 9 (* For monitoring *)
	???:PLC_CYCLE(reset_max_cycletime: reset_max, max_cycle_us => max_cycletime) => cycletime
NETWORK 10 (* Last line *)
	FALSE => init_1
_END_FBD_
(* the same logic as Structured Text *)
(* Network 1: see the listing above *)
(* Network 2 *)
RELAIS := TRUE;
(* Network 3 *)
IF init_e AND RELAIS THEN RELAIS_E := TRUE; END_IF;
(* Network 4: see the listing above *)
(* Network 5 *)
ga(ENABLE := TRUE, LEN := 200, MODE := 2);
(* Network 6: see the listing above *)
(* Network 7: see the listing above *)
(* Network 8: see the listing above *)
(* Network 9: see the listing above *)
(* Network 10 *)
init_1 := FALSE;
END_PROGRAM

(* POU INIT_MASTER_SLAVE_COMMUNICATION/SET_MASTER, FBD *)
PROGRAM SET_MASTER
VAR_INPUT
	init: BOOL := TRUE;
END_VAR
VAR_OUTPUT
	init_e:BOOL;
END_VAR

VAR
	Ssm1:SSC_SET_MASTER;
	prog_slave:DUMMY;
	com_intern_ok: BOOL;
END_VAR
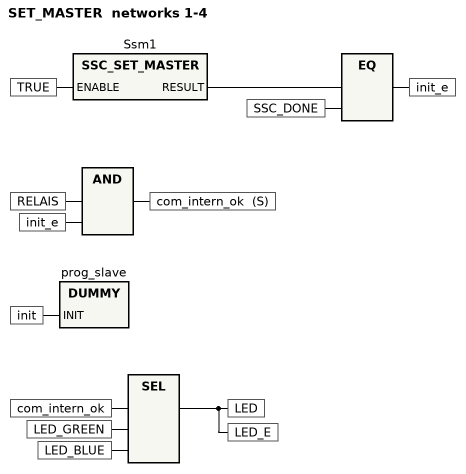
_FBD_ (* Function Block Diagram *)
NETWORK 1
	EQ(Ssm1:SSC_SET_MASTER(ENABLE: TRUE), SSC_DONE) => init_e
NETWORK 2
	AND(RELAIS, init_e) => S com_intern_ok
NETWORK 3
	prog_slave:DUMMY(INIT: init)
NETWORK 4
	SEL(com_intern_ok, LED_GREEN, LED_BLUE) => LED, LED_E
_END_FBD_
(* the same logic as Structured Text *)
(* Network 1 *)
Ssm1(ENABLE := TRUE);
init_e := Ssm1.RESULT = SSC_DONE;
(* Network 2 *)
IF RELAIS AND init_e THEN com_intern_ok := TRUE; END_IF;
(* Network 3 *)
prog_slave(INIT := init);
(* Network 4 *)
LED := SEL(com_intern_ok, LED_GREEN, LED_BLUE);
LED_E := LED;
END_PROGRAM

(* POU BOOTING, ST *)
PROGRAM BOOTING
VAR
	boot: BOOL;
	BLINK1: BLINK;


	ton1: TON;
	aa: BOOL;

	ton2: TON;
	aa1: BOOL;
	ton3: TON;
	ton4: TON;
END_VAR
IF aa THEN
	%MW0:=0;%MW2:=0;%MW4:=0;%MW6:=0;%MW8:=0;
	%MW10:=0;%MW12:=0;%MW14:=0;%MW16:=0;%MW18:=0;
	%MW20:=0;%MW22:=0;%MW24:=0;%MW26:=0;%MW28:=0;
	%MW30:=0;%MW32:=0;%MW34:=0;%MW36:=0;%MW38:=0;
	%MW40:=0;%MW42:=0;%MW44:=0;%MW46:=0;%MW48:=0;
	%MW50:=0;%MW52:=0;%MW54:=0;%MW56:=0;%MW58:=0;
	%MW60:=0;%MW62:=0;%MW64:=0;%MW66:=0;%MW68:=0;
	%MW70:=0;%MW72:=0;%MW74:=0;%MW76:=0;%MW78:=0;
	%MW80:=0;%MW82:=0;%MW84:=0;%MW86:=0;%MW88:=0;
	%MW90:=0;%MW92:=0;%MW94:=0;%MW96:=0;%MW98:=0;
END_IF

IF valve_act THEN
	IF	angle_x_offset=0		 				THEN angle_x_offset:=1000;				END_IF
	IF	angle_y_offset=0		 				THEN angle_y_offset:=1000;				END_IF
	IF	water_height_sign_L=0		 		THEN water_height_sign_L:=480;		END_IF
	IF	water_height_sign_H=0		 		THEN water_height_sign_H:=1557;		END_IF
	IF	foam_height_sign_L=0		 		THEN foam_height_sign_L:=480;		END_IF
	IF	foam_height_sign_H=0		 		THEN foam_height_sign_H:=1557;		END_IF
	IF	oil_pressure_0=0		 				THEN oil_pressure_0:=1000;			END_IF
	IF	oil_pressure_22=0		 			THEN oil_pressure_22:=13931;			END_IF
END_IF

IF NOT boot THEN
	boot:=TRUE;
	up_valve_ctl:=0;
	down_valve_ctl:=0;
	under_reset_ctl:=1;
	frequ_set:=1;
END_IF

IF NOT boot_set  AND NOT aa1 THEN
	ton3(IN:=(NOT boot_set ), PT:=T#3s  );
	IF ton3.q THEN
		boot_set:=1;
		aa1:=1;
		ton3(IN:=0);
	END_IF
END_IF

ton4(IN:=aa1, PT:=T#1s  );
IF ton4.q THEN
	boot_set:=0;
	ton2(IN:=0);
END_IF

ton2(IN:=NOT valve_act, PT:=T#6s  );
IF ton2.Q THEN 	valve_act:=1;END_IF

ton1(IN:=frequ_set, PT:=T#5s  );
IF ton1.Q THEN 	frequ_set:=0;END_IF

BLINK1(ENABLE:=TRUE , TIMELOW:= t#1s, TIMEHIGH:= t#1s , OUT=> down_com_sign);
END_PROGRAM

(* POU I_O_CONFIGURATION/CONF_IO_CR0200, FBD *)
PROGRAM CONF_IO_CR0200
VAR

END_VAR
VAR CONSTANT

	(*IN_NOMODE ==> all Bits 0*)
	IN_DIGITAL_H_ : BOOL := TRUE;	(*Bit 0*)
	IN_DIGITAL_L_ : BOOL:= TRUE;		(*Bit 1*)
	IN_CURRENT_ : BOOL := TRUE;	(*Bit 2*)
	IN_VOLTAGE10_ : BOOL := TRUE;	(*Bit 3*)
	IN_VOLTAGE30_ : BOOL := TRUE;	(*Bit 4*)
	IN_RATIO_ : BOOL := TRUE;			(*Bit 5*)
	IN_DIAGNOSTIC_ : BOOL := TRUE;	(*Bit 6*)

	IN_FAST_ : BOOL := TRUE;			(*Bit 7 *)

	(*OUT_NOMODE ==> all bits 0*)
	OUT_DIGITAL_H_ : BOOL := TRUE;						(*Bit 0*)
	OUT_DIGITAL_L_ : BOOL := TRUE;						(*Bit 1*)
	OUT_CURRENT_ : BOOL := TRUE;						(*Bit 2*)

	OUT_DIAGNOSTIC_ : BOOL := TRUE;					(*Bit 6*)
	OUT_OVERLOAD_PROTECTION_ : BOOL := TRUE;	(*Bit 7*)

END_VAR

VAR_INPUT
	INIT: BOOL;
END_VAR
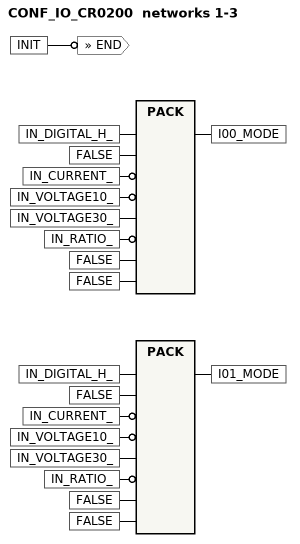
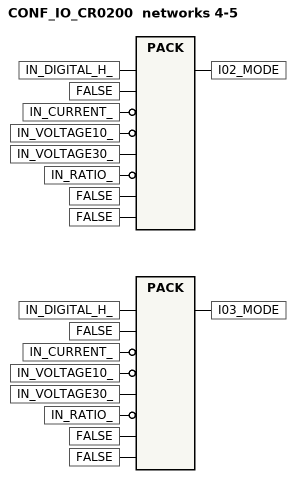
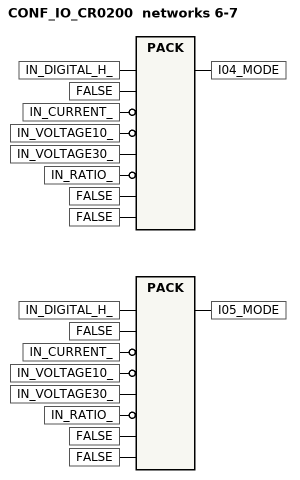
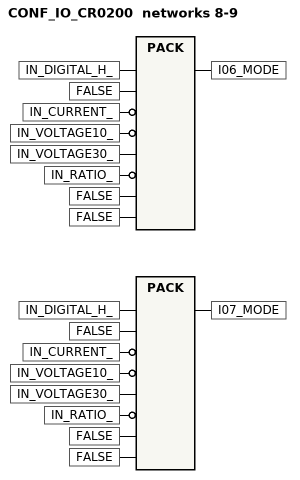
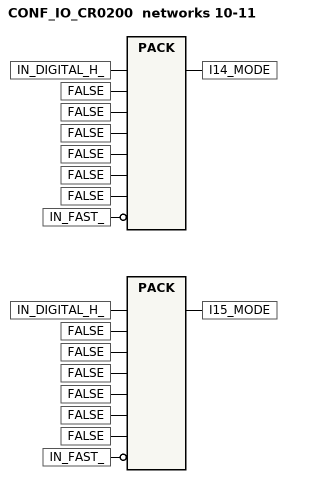
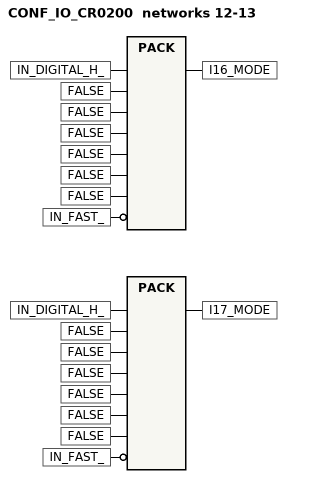
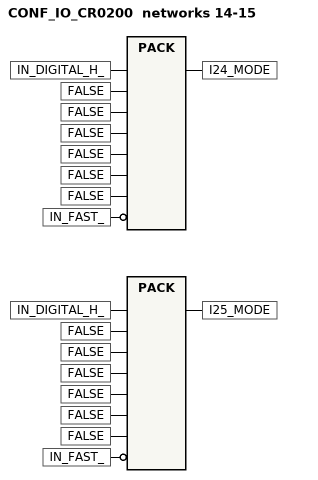
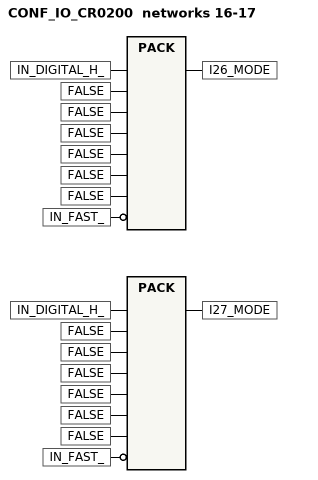
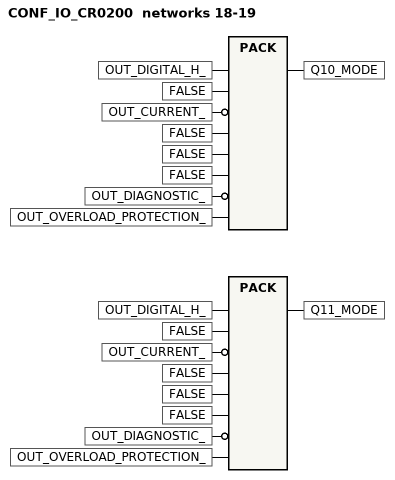
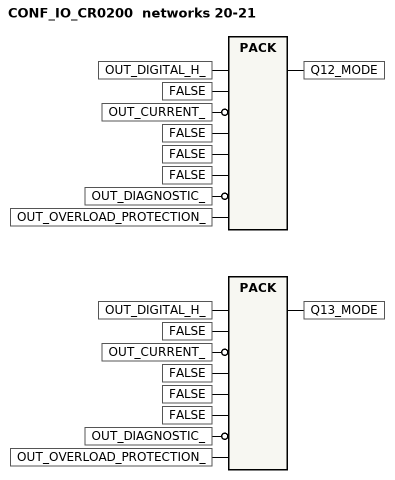
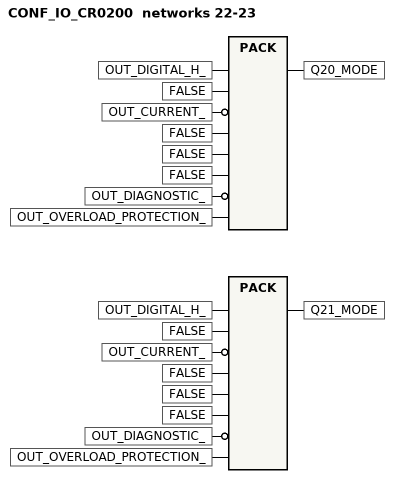
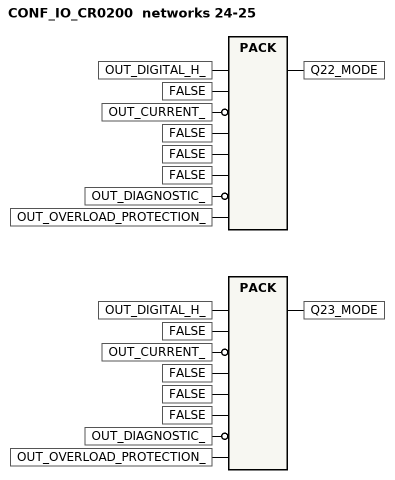
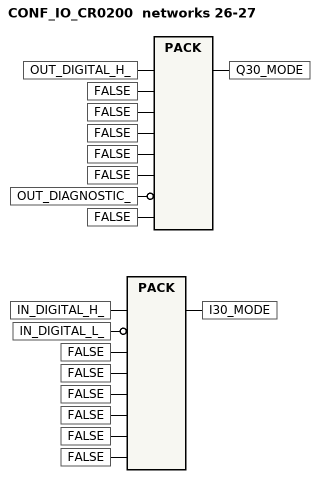
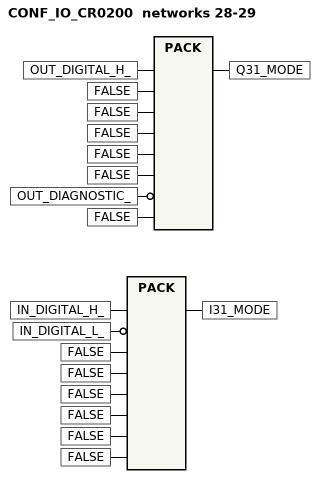
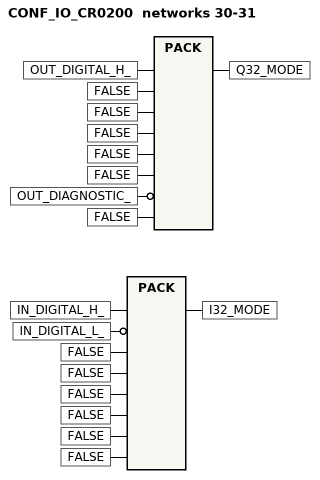
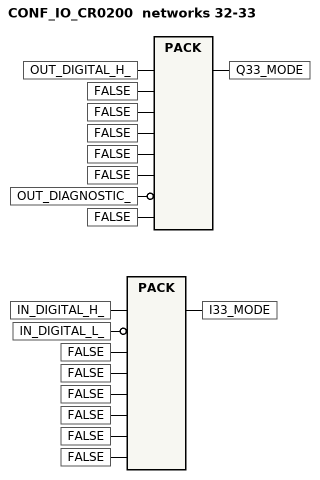
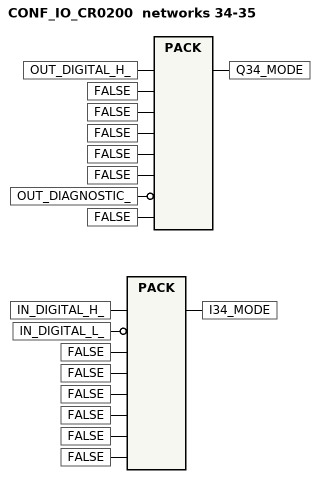
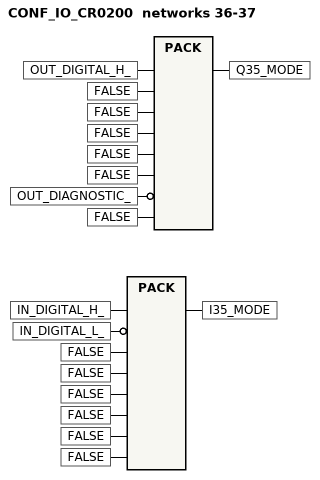
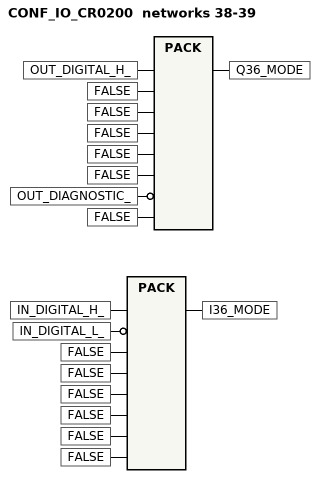
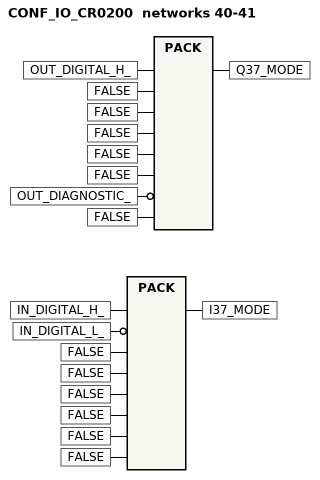
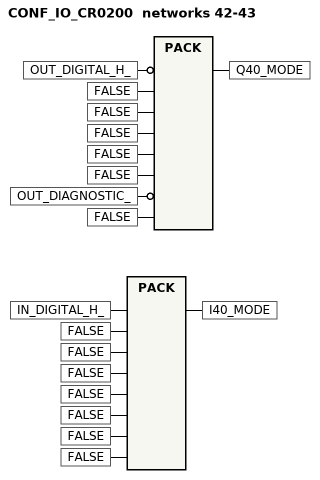
